LIN {X 0,Y 401.063,Z 357.189,A -85,B 0,C 180,E1 -11072.614,E2 -11072.614} C_VEL
LIN {X 0,Y 401.534,Z 344.039,A -85,B 0,C 180,E1 -11073.183,E2 -11073.183} C_VEL
LIN {X 0,Y 401.795,Z 330.677,A -85,B 0,C 180,E1 -11073.537,E2 -11073.537} C_VEL
LIN {X 0,Y 402.83,Z 248.147,A -85,B 0,C 180,E1 -11075.006,E2 -11075.006} C_VEL
LIN {X 0,Y 398.942,Z 226.266,A -85,B 0,C 180,E1 -11075.573,E2 -11075.573} C_VEL
LIN {X 0,Y 398.046,Z 222.975,A -85,B 0,C 180,E1 -11075.701,E2 -11075.701} C_VEL
LIN {X 0,Y 397.386,Z 219.987,A -85,B 0,C 180,E1 -11076.061,E2 -11076.061} C_VEL
LIN {X 0,Y 397.241,Z 220.003,A -85,B 0,C 180,E1 -11079.163,E2 -11079.163} C_VEL
LIN {X 0,Y 397.225,Z 220.006,A -85,B 0,C 180,E1 -11082.259,E2 -11082.259} C_VEL
LIN {X 0,Y 397.184,Z 220.008,A -85,B 0,C 180,E1 -11085.393,E2 -11085.393} C_VEL
LIN {X 0,Y 397.167,Z 220.014,A -85,B 0,C 180,E1 -11088.574,E2 -11088.574} C_VEL
LIN {X 0,Y 397.102,Z 220.021,A -85,B 0,C 180,E1 -11091.819,E2 -11091.819} C_VEL
LIN {X 0,Y 397.11,Z 220.018,A -85,B 0,C 180,E1 -11095.136,E2 -11095.136} C_VEL
LIN {X 0,Y 397.071,Z 220.024,A -85,B 0,C 180,E1 -11098.549,E2 -11098.549} C_VEL
LIN {X 0,Y 397.086,Z 220.023,A -85,B 0,C 180,E1 -11101.836,E2 -11101.836} C_VEL
LIN {X 0,Y 397.123,Z 220.017,A -85,B 0,C 180,E1 -11104.495,E2 -11104.495} C_VEL
LIN {X 0,Y 397.093,Z 220.021,A -85,B 0,C 180,E1 -11108.277,E2 -11108.277} C_VEL
LIN {X 0,Y 397.056,Z 220.027,A -85,B 0,C 180,E1 -11111.976,E2 -11111.976} C_VEL
LIN {X 0,Y 397.09,Z 220.023,A -85,B 0,C 180,E1 -11115.07,E2 -11115.07} C_VEL
LIN {X 0,Y 397.056,Z 220.025,A -85,B 0,C 180,E1 -11118.024,E2 -11118.024} C_VEL
LIN {X 0,Y 397.092,Z 220.023,A -85,B 0,C 180,E1 -11121.147,E2 -11121.147} C_VEL
LIN {X 0,Y 397.095,Z 220.021,A -85,B 0,C 180,E1 -11124.503,E2 -11124.503} C_VEL
LIN {X 0,Y 397.077,Z 220.022,A -85,B 0,C 180,E1 -11127.928,E2 -11127.928} C_VEL
LIN {X 0,Y 397.119,Z 220.018,A -85,B 0,C 180,E1 -11130.295,E2 -11130.295} C_VEL
LIN {X 0,Y 397.076,Z 220.022,A -85,B 0,C 180,E1 -11133.737,E2 -11133.737} C_VEL
LIN {X 0,Y 397.16,Z 220.084,A -85,B 0,C 180,E1 -11137.363,E2 -11137.363} C_VEL
LIN {X 0,Y 398.579,Z 228.682,A -85,B 0,C 180,E1 -11139.62,E2 -11139.62} C_VEL
LIN {X 0,Y 398.602,Z 228.95,A -85,B 0,C 180,E1 -11139.688,E2 -11139.688} C_VEL
LIN {X 0,Y 402.439,Z 249.604,A -85,B 0,C 180,E1 -11140.323,E2 -11140.323} C_VEL
LIN {X 0,Y 400.599,Z 337.679,A -85,B 0,C 180,E1 -11142.318,E2 -11142.318} C_VEL
LIN {X 0,Y 400.213,Z 351.101,A -85,B 0,C 180,E1 -11142.828,E2 -11142.828} C_VEL
LIN {X 0,Y 399.791,Z 363.98,A -85,B 0,C 180,E1 -11143.533,E2 -11143.533} C_VEL
LIN {X 0,Y 399.118,Z 376.314,A -85,B 0,C 180,E1 -11144.423,E2 -11144.423} C_VEL
LIN {X 0,Y 398.537,Z 387.459,A -85,B 0,C 180,E1 -11145.446,E2 -11145.446} C_VEL
LIN {X 0,Y 397.965,Z 398.566,A -85,B 0,C 180,E1 -11146.727,E2 -11146.727} C_VEL
LIN {X 0,Y 397.414,Z 407.599,A -85,B 0,C 180,E1 -11148.007,E2 -11148.007} C_VEL
LIN {X 0,Y 396.89,Z 416.341,A -85,B 0,C 180,E1 -11149.542,E2 -11149.542} C_VEL
LIN {X 0,Y 396.494,Z 423.36,A -85,B 0,C 180,E1 -11151.077,E2 -11151.077} C_VEL
LIN {X 0,Y 396.215,Z 429.747,A -85,B 0,C 180,E1 -11152.867,E2 -11152.867} C_VEL
LIN {X 0,Y 396.072,Z 433.874,A -85,B 0,C 180,E1 -11154.399,E2 -11154.399} C_VEL
LIN {X 0,Y 395.924,Z 436.902,A -85,B 0,C 180,E1 -11155.928,E2 -11155.928} C_VEL
LIN {X 0,Y 395.946,Z 438.34,A -85,B 0,C 180,E1 -11156.947,E2 -11156.947} C_VEL
LIN {X 0,Y 395.921,Z 439.365,A -85,B 0,C 180,E1 -11157.965,E2 -11157.965} C_VEL
LIN {X 0,Y 395.851,Z 439.942,A -85,B 0,C 180,E1 -11158.982,E2 -11158.982} C_VEL
LIN {X 0,Y 395.86,Z 440.071,A -85,B 0,C 180,E1 -11160,E2 -11160} C_VEL
LIN {X 0,Y 395.915,Z 439.79,A -85,B 0,C 180,E1 -11161.017,E2 -11161.017} C_VEL
LIN {X 0,Y 396.011,Z 439.092,A -85,B 0,C 180,E1 -11162.034,E2 -11162.034} C_VEL
LIN {X 0,Y 396.188,Z 437.92,A -85,B 0,C 180,E1 -11163.05,E2 -11163.05} C_VEL
LIN {X 0,Y 396.462,Z 435.363,A -85,B 0,C 180,E1 -11164.575,E2 -11164.575} C_VEL
LIN {X 0,Y 396.56,Z 431.768,A -85,B 0,C 180,E1 -11166.104,E2 -11166.104} C_VEL
LIN {X 0,Y 397.232,Z 426.428,A -85,B 0,C 180,E1 -11167.782,E2 -11167.782} C_VEL
LIN {X 0,Y 397.81,Z 419.827,A -85,B 0,C 180,E1 -11169.405,E2 -11169.405} C_VEL
LIN {X 0,Y 398.625,Z 411.939,A -85,B 0,C 180,E1 -11170.925,E2 -11170.925} C_VEL
LIN {X 0,Y 399.377,Z 403.929,A -85,B 0,C 180,E1 -11172.191,E2 -11172.191} C_VEL
LIN {X 0,Y 400.233,Z 394.193,A -85,B 0,C 180,E1 -11173.454,E2 -11173.454} C_VEL
LIN {X 0,Y 401.25,Z 383.309,A -85,B 0,C 180,E1 -11174.583,E2 -11174.583} C_VEL
LIN {X 0,Y 402.03,Z 372.326,A -85,B 0,C 180,E1 -11175.504,E2 -11175.504} C_VEL
LIN {X 0,Y 402.835,Z 360.204,A -85,B 0,C 180,E1 -11176.299,E2 -11176.299} C_VEL
LIN {X 0,Y 403.424,Z 346.397,A -85,B 0,C 180,E1 -11176.965,E2 -11176.965} C_VEL
LIN {X 0,Y 403.901,Z 332.803,A -85,B 0,C 180,E1 -11177.401,E2 -11177.401} C_VEL
LIN {X 0,Y 406.565,Z 263.883,A -85,B 0,C 180,E1 -11179.143,E2 -11179.143} C_VEL
LIN {X 0,Y 406.93,Z 252.02,A -85,B 0,C 180,E1 -11179.466,E2 -11179.466} C_VEL
LIN {X 0,Y 404.708,Z 243.879,A -85,B 0,C 180,E1 -11179.902,E2 -11179.902} C_VEL
LIN {X 0,Y 401.099,Z 235.68,A -85,B 0,C 180,E1 -11180.482,E2 -11180.482} C_VEL
LIN {X 0,Y 400.343,Z 233.798,A -85,B 0,C 180,E1 -11180.618,E2 -11180.618} C_VEL
LIN {X 0,Y 398.311,Z 224.634,A -85,B 0,C 180,E1 -11183.943,E2 -11183.943} C_VEL
LIN {X 0,Y 397.149,Z 220.017,A -85,B 0,C 180,E1 -11185.833,E2 -11185.833} C_VEL
LIN {X 0,Y 397.128,Z 220.019,A -85,B 0,C 180,E1 -11188.543,E2 -11188.543} C_VEL
LIN {X 0,Y 397.084,Z 220.024,A -85,B 0,C 180,E1 -11192.071,E2 -11192.071} C_VEL
LIN {X 0,Y 397.125,Z 220.018,A -85,B 0,C 180,E1 -11195.503,E2 -11195.503} C_VEL
LIN {X 0,Y 397.135,Z 220.015,A -85,B 0,C 180,E1 -11198.861,E2 -11198.861} C_VEL
LIN {X 0,Y 397.073,Z 220.024,A -85,B 0,C 180,E1 -11202.267,E2 -11202.267} C_VEL
LIN {X 0,Y 397.091,Z 220.021,A -85,B 0,C 180,E1 -11205.068,E2 -11205.068} C_VEL
LIN {X 0,Y 397.067,Z 220.025,A -85,B 0,C 180,E1 -11208.021,E2 -11208.021} C_VEL
LIN {X 0,Y 397.128,Z 220.016,A -85,B 0,C 180,E1 -11211.139,E2 -11211.139} C_VEL
LIN {X 0,Y 397.123,Z 220.019,A -85,B 0,C 180,E1 -11214.496,E2 -11214.496} C_VEL
LIN {X 0,Y 397.114,Z 220.1,A -85,B 0,C 180,E1 -11217.481,E2 -11217.481} C_VEL
LIN {X 0,Y 399.599,Z 229.04,A -85,B 0,C 180,E1 -11220.497,E2 -11220.497} C_VEL
LIN {X 0,Y 401.612,Z 238.359,A -85,B 0,C 180,E1 -11223.186,E2 -11223.186} C_VEL
LIN {X 0,Y 402.307,Z 242.854,A -85,B 0,C 180,E1 -11224.381,E2 -11224.381} C_VEL
LIN {X 0,Y 400.576,Z 257.062,A -85,B 0,C 180,E1 -11227.566,E2 -11227.566} C_VEL
LIN {X 0,Y 400.165,Z 260.831,A -85,B 0,C 180,E1 -11228.382,E2 -11228.382} C_VEL
LIN {X 0,Y 403.739,Z 277.867,A -85,B 0,C 180,E1 -11229.213,E2 -11229.213} C_VEL
LIN {X 0,Y 405.673,Z 291.849,A -85,B 0,C 180,E1 -11229.776,E2 -11229.776} C_VEL
LIN {X 0,Y 405.744,Z 299.247,A -85,B 0,C 180,E1 -11229.996,E2 -11229.996} C_VEL
LIN {X 0,Y 403.15,Z 373.349,A -85,B 0,C 180,E1 -11231.875,E2 -11231.875} C_VEL
LIN {X 0,Y 402.379,Z 386.533,A -85,B 0,C 180,E1 -11232.398,E2 -11232.398} C_VEL
LIN {X 0,Y 401.432,Z 398.799,A -85,B 0,C 180,E1 -11233.078,E2 -11233.078} C_VEL
LIN {X 0,Y 400.503,Z 410.917,A -85,B 0,C 180,E1 -11233.955,E2 -11233.955} C_VEL
LIN {X 0,Y 399.499,Z 421.992,A -85,B 0,C 180,E1 -11234.96,E2 -11234.96} C_VEL
LIN {X 0,Y 398.415,Z 433.079,A -85,B 0,C 180,E1 -11236.22,E2 -11236.22} C_VEL
LIN {X 0,Y 397.788,Z 442.22,A -85,B 0,C 180,E1 -11237.5,E2 -11237.5} C_VEL
LIN {X 0,Y 397.011,Z 449.795,A -85,B 0,C 180,E1 -11238.77,E2 -11238.77} C_VEL
LIN {X 0,Y 396.51,Z 457.268,A -85,B 0,C 180,E1 -11240.305,E2 -11240.305} C_VEL
LIN {X 0,Y 396.148,Z 463.253,A -85,B 0,C 180,E1 -11241.84,E2 -11241.84} C_VEL
LIN {X 0,Y 395.896,Z 467.98,A -85,B 0,C 180,E1 -11243.373,E2 -11243.373} C_VEL
LIN {X 0,Y 395.83,Z 471.57,A -85,B 0,C 180,E1 -11244.906,E2 -11244.906} C_VEL
LIN {X 0,Y 395.781,Z 473.371,A -85,B 0,C 180,E1 -11245.926,E2 -11245.926} C_VEL
LIN {X 0,Y 395.766,Z 474.741,A -85,B 0,C 180,E1 -11246.945,E2 -11246.945} C_VEL
LIN {X 0,Y 395.856,Z 475.636,A -85,B 0,C 180,E1 -11247.964,E2 -11247.964} C_VEL
LIN {X 0,Y 395.832,Z 476.09,A -85,B 0,C 180,E1 -11248.982,E2 -11248.982} C_VEL
LIN {X 0,Y 395.832,Z 476.126,A -85,B 0,C 180,E1 -11249.999,E2 -11249.999} C_VEL
LIN {X 0,Y 395.832,Z 475.723,A -85,B 0,C 180,E1 -11251.016,E2 -11251.016} C_VEL
LIN {X 0,Y 395.884,Z 474.843,A -85,B 0,C 180,E1 -11252.034,E2 -11252.034} C_VEL
LIN {X 0,Y 395.804,Z 471.823,A -85,B 0,C 180,E1 -11254.072,E2 -11254.072} C_VEL
LIN {X 0,Y 395.825,Z 468.629,A -85,B 0,C 180,E1 -11255.805,E2 -11255.805} C_VEL
LIN {X 0,Y 396.05,Z 463.765,A -85,B 0,C 180,E1 -11257.647,E2 -11257.647} C_VEL
LIN {X 0,Y 396.396,Z 457.411,A -85,B 0,C 180,E1 -11259.438,E2 -11259.438} C_VEL
LIN {X 0,Y 396.877,Z 450.497,A -85,B 0,C 180,E1 -11260.973,E2 -11260.973} C_VEL
LIN {X 0,Y 397.698,Z 441.836,A -85,B 0,C 180,E1 -11262.501,E2 -11262.501} C_VEL
LIN {X 0,Y 398.48,Z 432.076,A -85,B 0,C 180,E1 -11263.892,E2 -11263.892} C_VEL
LIN {X 0,Y 399.464,Z 421.988,A -85,B 0,C 180,E1 -11265.039,E2 -11265.039} C_VEL
LIN {X 0,Y 400.44,Z 410.878,A -85,B 0,C 180,E1 -11266.046,E2 -11266.046} C_VEL
LIN {X 0,Y 401.396,Z 398.415,A -85,B 0,C 180,E1 -11266.922,E2 -11266.922} C_VEL
LIN {X 0,Y 402.198,Z 385.528,A -85,B 0,C 180,E1 -11267.575,E2 -11267.575} C_VEL
LIN {X 0,Y 402.857,Z 372.832,A -85,B 0,C 180,E1 -11268.004,E2 -11268.004} C_VEL
LIN {X 0,Y 403.564,Z 325.155,A -85,B 0,C 180,E1 -11268.907,E2 -11268.907} C_VEL
LIN {X 0,Y 403.921,Z 293.473,A -85,B 0,C 180,E1 -11269.491,E2 -11269.491} C_VEL
LIN {X 0,Y 400.513,Z 269.928,A -85,B 0,C 180,E1 -11270.146,E2 -11270.146} C_VEL
LIN {X 0,Y 398.784,Z 259.631,A -85,B 0,C 180,E1 -11270.458,E2 -11270.458} C_VEL
LIN {X 0,Y 400.229,Z 239.999,A -85,B 0,C 180,E1 -11274.394,E2 -11274.394} C_VEL
LIN {X 0,Y 400.31,Z 236.077,A -85,B 0,C 180,E1 -11275.196,E2 -11275.196} C_VEL
LIN {X 0,Y 397.701,Z 222.504,A -85,B 0,C 180,E1 -11278.168,E2 -11278.168} C_VEL
LIN {X 0,Y 397.184,Z 220.012,A -85,B 0,C 180,E1 -11278.754,E2 -11278.754} C_VEL
LIN {X 0,Y 397.075,Z 220.011,A -85,B 0,C 180,E1 -11282.07,E2 -11282.07} C_VEL
LIN {X 0,Y 397.114,Z 220.009,A -85,B 0,C 180,E1 -11285.502,E2 -11285.502} C_VEL
LIN {X 0,Y 397.087,Z 220.014,A -85,B 0,C 180,E1 -11288.854,E2 -11288.854} C_VEL
LIN {X 0,Y 397.055,Z 220.02,A -85,B 0,C 180,E1 -11292.267,E2 -11292.267} C_VEL
LIN {X 0,Y 397.079,Z 220.02,A -85,B 0,C 180,E1 -11295.068,E2 -11295.068} C_VEL
LIN {X 0,Y 397.046,Z 220.014,A -85,B 0,C 180,E1 -11298.022,E2 -11298.022} C_VEL
LIN {X 0,Y 397.085,Z 220.02,A -85,B 0,C 180,E1 -11301.723,E2 -11301.723} C_VEL
LIN {X 0,Y 397.117,Z 220.01,A -85,B 0,C 180,E1 -11305.506,E2 -11305.506} C_VEL
LIN {X 0,Y 397.069,Z 220.014,A -85,B 0,C 180,E1 -11309.117,E2 -11309.117} C_VEL
LIN {X 0,Y 397.054,Z 220.013,A -85,B 0,C 180,E1 -11312.251,E2 -11312.251} C_VEL
LIN {X 0,Y 397.093,Z 220.02,A -85,B 0,C 180,E1 -11314.864,E2 -11314.864} C_VEL
LIN {X 0,Y 397.085,Z 219.996,A -85,B 0,C 180,E1 -11318.181,E2 -11318.181} C_VEL
LIN {X 0,Y 397.147,Z 220.011,A -85,B 0,C 180,E1 -11321.426,E2 -11321.426} C_VEL
LIN {X 0,Y 397.159,Z 219.999,A -85,B 0,C 180,E1 -11324.607,E2 -11324.607} C_VEL
LIN {X 0,Y 397.209,Z 219.995,A -85,B 0,C 180,E1 -11327.742,E2 -11327.742} C_VEL
LIN {X 0,Y 397.225,Z 220.004,A -85,B 0,C 180,E1 -11330.838,E2 -11330.838} C_VEL
LIN {X 0,Y 397.306,Z 219.977,A -85,B 0,C 180,E1 -11333.908,E2 -11333.908} C_VEL
LIN {X 0,Y 397.437,Z 219.974,A -85,B 0,C 180,E1 -11337.973,E2 -11337.973} C_VEL
LIN {X 0,Y 397.364,Z 219.974,A -85,B 0,C 180,E1 -11341.014,E2 -11341.014} C_VEL
LIN {X 0,Y 397.321,Z 219.969,A -85,B 0,C 180,E1 -11343.042,E2 -11343.042} C_VEL
LIN {X 0,Y 397.334,Z 219.985,A -85,B 0,C 180,E1 -11346.643,E2 -11346.643} C_VEL
LIN {X 0,Y 397.244,Z 219.989,A -85,B 0,C 180,E1 -11349.162,E2 -11349.162} C_VEL
LIN {X 0,Y 397.21,Z 220,A -85,B 0,C 180,E1 -11352.259,E2 -11352.259} C_VEL
LIN {X 0,Y 397.171,Z 220.008,A -85,B 0,C 180,E1 -11355.393,E2 -11355.393} C_VEL
LIN {X 0,Y 397.15,Z 220.005,A -85,B 0,C 180,E1 -11358.574,E2 -11358.574} C_VEL
LIN {X 0,Y 397.102,Z 220.017,A -85,B 0,C 180,E1 -11361.819,E2 -11361.819} C_VEL
LIN {X 0,Y 397.146,Z 220.011,A -85,B 0,C 180,E1 -11365.513,E2 -11365.513} C_VEL
LIN {X 0,Y 397.116,Z 220.011,A -85,B 0,C 180,E1 -11368.545,E2 -11368.545} C_VEL
LIN {X 0,Y 397.073,Z 220.023,A -85,B 0,C 180,E1 -11372.073,E2 -11372.073} C_VEL
LIN {X 0,Y 397.115,Z 220.021,A -85,B 0,C 180,E1 -11375.505,E2 -11375.505} C_VEL
LIN {X 0,Y 397.129,Z 220.013,A -85,B 0,C 180,E1 -11378.863,E2 -11378.863} C_VEL
LIN {X 0,Y 397.067,Z 220.019,A -85,B 0,C 180,E1 -11382.268,E2 -11382.268} C_VEL
LIN {X 0,Y 397.088,Z 220.02,A -85,B 0,C 180,E1 -11385.069,E2 -11385.069} C_VEL
LIN {X 0,Y 397.065,Z 220.022,A -85,B 0,C 180,E1 -11388.022,E2 -11388.022} C_VEL
LIN {X 0,Y 397.129,Z 220.017,A -85,B 0,C 180,E1 -11391.14,E2 -11391.14} C_VEL
LIN {X 0,Y 397.189,Z 220.178,A -85,B 0,C 180,E1 -11394.835,E2 -11394.835} C_VEL
LIN {X 0,Y 398.26,Z 223.723,A -85,B 0,C 180,E1 -11395.233,E2 -11395.233} C_VEL
LIN {X 0,Y 402.441,Z 234.001,A -85,B 0,C 180,E1 -11395.7,E2 -11395.7} C_VEL
LIN {X 0,Y 405.169,Z 249.064,A -85,B 0,C 180,E1 -11396.158,E2 -11396.158} C_VEL
LIN {X 0,Y 403.759,Z 336.274,A -85,B 0,C 180,E1 -11397.751,E2 -11397.751} C_VEL
LIN {X 0,Y 403.309,Z 349.643,A -85,B 0,C 180,E1 -11398.19,E2 -11398.19} C_VEL
LIN {X 0,Y 402.684,Z 362.586,A -85,B 0,C 180,E1 -11398.845,E2 -11398.845} C_VEL
LIN {X 0,Y 401.924,Z 374.716,A -85,B 0,C 180,E1 -11399.676,E2 -11399.676} C_VEL
LIN {X 0,Y 400.96,Z 386.467,A -85,B 0,C 180,E1 -11400.728,E2 -11400.728} C_VEL
LIN {X 0,Y 399.92,Z 397.351,A -85,B 0,C 180,E1 -11401.961,E2 -11401.961} C_VEL
LIN {X 0,Y 399.022,Z 406.833,A -85,B 0,C 180,E1 -11403.313,E2 -11403.313} C_VEL
LIN {X 0,Y 398.081,Z 415.911,A -85,B 0,C 180,E1 -11404.932,E2 -11404.932} C_VEL
LIN {X 0,Y 397.365,Z 423.026,A -85,B 0,C 180,E1 -11406.539,E2 -11406.539} C_VEL
LIN {X 0,Y 396.787,Z 428.692,A -85,B 0,C 180,E1 -11408.165,E2 -11408.165} C_VEL
LIN {X 0,Y 396.333,Z 433.595,A -85,B 0,C 180,E1 -11410.024,E2 -11410.024} C_VEL
LIN {X 0,Y 396.04,Z 436.166,A -85,B 0,C 180,E1 -11411.373,E2 -11411.373} C_VEL
LIN {X 0,Y 395.884,Z 437.703,A -85,B 0,C 180,E1 -11412.436,E2 -11412.436} C_VEL
LIN {X 0,Y 395.822,Z 438.749,A -85,B 0,C 180,E1 -11413.497,E2 -11413.497} C_VEL
LIN {X 0,Y 395.754,Z 439.384,A -85,B 0,C 180,E1 -11414.552,E2 -11414.552} C_VEL
LIN {X 0,Y 395.717,Z 439.618,A -85,B 0,C 180,E1 -11415.604,E2 -11415.604} C_VEL
LIN {X 0,Y 395.783,Z 438.843,A -85,B 0,C 180,E1 -11417.595,E2 -11417.595} C_VEL
LIN {X 0,Y 395.809,Z 437.743,A -85,B 0,C 180,E1 -11418.738,E2 -11418.738} C_VEL
LIN {X 0,Y 395.835,Z 436.284,A -85,B 0,C 180,E1 -11419.774,E2 -11419.774} C_VEL
LIN {X 0,Y 396.083,Z 433.264,A -85,B 0,C 180,E1 -11421.327,E2 -11421.327} C_VEL
LIN {X 0,Y 396.402,Z 428.325,A -85,B 0,C 180,E1 -11423.15,E2 -11423.15} C_VEL
LIN {X 0,Y 396.707,Z 421.962,A -85,B 0,C 180,E1 -11424.919,E2 -11424.919} C_VEL
LIN {X 0,Y 397.295,Z 414.866,A -85,B 0,C 180,E1 -11426.451,E2 -11426.451} C_VEL
LIN {X 0,Y 397.977,Z 406.078,A -85,B 0,C 180,E1 -11427.977,E2 -11427.977} C_VEL
LIN {X 0,Y 398.722,Z 395.987,A -85,B 0,C 180,E1 -11429.37,E2 -11429.37} C_VEL
LIN {X 0,Y 399.486,Z 385.754,A -85,B 0,C 180,E1 -11430.505,E2 -11430.505} C_VEL
LIN {X 0,Y 400.238,Z 374.372,A -85,B 0,C 180,E1 -11431.51,E2 -11431.51} C_VEL
LIN {X 0,Y 400.524,Z 369.63,A -85,B 0,C 180,E1 -11431.859,E2 -11431.859} C_VEL
LIN {X 0,Y 400.19,Z 364.343,A -85,B 0,C 180,E1 -11432.233,E2 -11432.233} C_VEL
LIN {X 0,Y 397.799,Z 355.633,A -85,B 0,C 180,E1 -11432.82,E2 -11432.82} C_VEL
LIN {X 0,Y 395.32,Z 346.674,A -85,B 0,C 180,E1 -11433.318,E2 -11433.318} C_VEL
LIN {X 0,Y 394.766,Z 340.998,A -85,B 0,C 180,E1 -11433.539,E2 -11433.539} C_VEL
LIN {X 0,Y 395.025,Z 326.392,A -85,B 0,C 180,E1 -11433.876,E2 -11433.876} C_VEL
LIN {X 0,Y 395.954,Z 248.651,A -85,B 0,C 180,E1 -11435.284,E2 -11435.284} C_VEL
LIN {X 0,Y 392.347,Z 228.274,A -85,B 0,C 180,E1 -11435.822,E2 -11435.822} C_VEL
LIN {X 0,Y 390.875,Z 223.251,A -85,B 0,C 180,E1 -11436,E2 -11436} C_VEL
LIN {X 0,Y 390.309,Z 220.868,A -85,B 0,C 180,E1 -11436.268,E2 -11436.268} C_VEL
LIN {X 0,Y 390.198,Z 220.879,A -85,B 0,C 180,E1 -11439.33,E2 -11439.33} C_VEL
LIN {X 0,Y 390.176,Z 220.884,A -85,B 0,C 180,E1 -11442.484,E2 -11442.484} C_VEL
LIN {X 0,Y 390.145,Z 220.885,A -85,B 0,C 180,E1 -11445.678,E2 -11445.678} C_VEL
LIN {X 0,Y 390.111,Z 220.89,A -85,B 0,C 180,E1 -11448.923,E2 -11448.923} C_VEL
LIN {X 0,Y 390.042,Z 220.901,A -85,B 0,C 180,E1 -11452.235,E2 -11452.235} C_VEL
LIN {X 0,Y 390.056,Z 220.899,A -85,B 0,C 180,E1 -11455.723,E2 -11455.723} C_VEL
LIN {X 0,Y 390.031,Z 220.899,A -85,B 0,C 180,E1 -11459.113,E2 -11459.113} C_VEL
LIN {X 0,Y 390.047,Z 220.897,A -85,B 0,C 180,E1 -11462.722,E2 -11462.722} C_VEL
LIN {X 0,Y 390.049,Z 220.9,A -85,B 0,C 180,E1 -11465.823,E2 -11465.823} C_VEL
LIN {X 0,Y 390.04,Z 220.9,A -85,B 0,C 180,E1 -11469.212,E2 -11469.212} C_VEL
LIN {X 0,Y 390.035,Z 220.899,A -85,B 0,C 180,E1 -11472.372,E2 -11472.372} C_VEL
LIN {X 0,Y 390.046,Z 220.901,A -85,B 0,C 180,E1 -11475.354,E2 -11475.354} C_VEL
LIN {X 0,Y 390.019,Z 220.901,A -85,B 0,C 180,E1 -11478.185,E2 -11478.185} C_VEL
LIN {X 0,Y 390.059,Z 220.899,A -85,B 0,C 180,E1 -11480.903,E2 -11480.903} C_VEL
LIN {X 0,Y 390.066,Z 220.898,A -85,B 0,C 180,E1 -11484.791,E2 -11484.791} C_VEL
LIN {X 0,Y 390.031,Z 220.899,A -85,B 0,C 180,E1 -11487.878,E2 -11487.878} C_VEL
LIN {X 0,Y 390.027,Z 220.903,A -85,B 0,C 180,E1 -11490.887,E2 -11490.887} C_VEL
LIN {X 0,Y 390.067,Z 220.897,A -85,B 0,C 180,E1 -11494.378,E2 -11494.378} C_VEL
LIN {X 0,Y 390.108,Z 220.937,A -85,B 0,C 180,E1 -11497.211,E2 -11497.211} C_VEL
LIN {X 0,Y 391.556,Z 229.176,A -85,B 0,C 180,E1 -11499.409,E2 -11499.409} C_VEL
LIN {X 0,Y 395.558,Z 250.268,A -85,B 0,C 180,E1 -11500.09,E2 -11500.09} C_VEL
LIN {X 0,Y 393.638,Z 337.821,A -85,B 0,C 180,E1 -11502.129,E2 -11502.129} C_VEL
LIN {X 0,Y 393.23,Z 351.232,A -85,B 0,C 180,E1 -11502.647,E2 -11502.647} C_VEL
LIN {X 0,Y 392.788,Z 364.143,A -85,B 0,C 180,E1 -11503.364,E2 -11503.364} C_VEL
LIN {X 0,Y 392.107,Z 376.495,A -85,B 0,C 180,E1 -11504.27,E2 -11504.27} C_VEL
LIN {X 0,Y 391.519,Z 387.674,A -85,B 0,C 180,E1 -11505.312,E2 -11505.312} C_VEL
LIN {X 0,Y 390.93,Z 398.804,A -85,B 0,C 180,E1 -11506.617,E2 -11506.617} C_VEL
LIN {X 0,Y 390.296,Z 408.668,A -85,B 0,C 180,E1 -11508.048,E2 -11508.048} C_VEL
LIN {X 0,Y 389.793,Z 417.273,A -85,B 0,C 180,E1 -11509.612,E2 -11509.612} C_VEL
LIN {X 0,Y 389.392,Z 424.199,A -85,B 0,C 180,E1 -11511.175,E2 -11511.175} C_VEL
LIN {X 0,Y 389.131,Z 429.692,A -85,B 0,C 180,E1 -11512.737,E2 -11512.737} C_VEL
LIN {X 0,Y 388.998,Z 433.93,A -85,B 0,C 180,E1 -11514.297,E2 -11514.297} C_VEL
LIN {X 0,Y 388.846,Z 437.056,A -85,B 0,C 180,E1 -11515.854,E2 -11515.854} C_VEL
LIN {X 0,Y 388.847,Z 438.54,A -85,B 0,C 180,E1 -11516.892,E2 -11516.892} C_VEL
LIN {X 0,Y 388.837,Z 439.608,A -85,B 0,C 180,E1 -11517.928,E2 -11517.928} C_VEL
LIN {X 0,Y 388.78,Z 440.262,A -85,B 0,C 180,E1 -11518.964,E2 -11518.964} C_VEL
LIN {X 0,Y 388.785,Z 440.443,A -85,B 0,C 180,E1 -11520,E2 -11520} C_VEL
LIN {X 0,Y 388.841,Z 440.204,A -85,B 0,C 180,E1 -11521.035,E2 -11521.035} C_VEL
LIN {X 0,Y 388.945,Z 439.556,A -85,B 0,C 180,E1 -11522.071,E2 -11522.071} C_VEL
LIN {X 0,Y 389.131,Z 438.453,A -85,B 0,C 180,E1 -11523.106,E2 -11523.106} C_VEL
LIN {X 0,Y 389.328,Z 436.899,A -85,B 0,C 180,E1 -11524.141,E2 -11524.141} C_VEL
LIN {X 0,Y 389.551,Z 433.741,A -85,B 0,C 180,E1 -11525.694,E2 -11525.694} C_VEL
LIN {X 0,Y 389.97,Z 429.466,A -85,B 0,C 180,E1 -11527.247,E2 -11527.247} C_VEL
LIN {X 0,Y 390.591,Z 423.97,A -85,B 0,C 180,E1 -11528.797,E2 -11528.797} C_VEL
LIN {X 0,Y 391.311,Z 417.093,A -85,B 0,C 180,E1 -11530.346,E2 -11530.346} C_VEL
LIN {X 0,Y 392.176,Z 408.454,A -85,B 0,C 180,E1 -11531.893,E2 -11531.893} C_VEL
LIN {X 0,Y 393.015,Z 399.655,A -85,B 0,C 180,E1 -11533.179,E2 -11533.179} C_VEL
LIN {X 0,Y 394.111,Z 388.807,A -85,B 0,C 180,E1 -11534.457,E2 -11534.457} C_VEL
LIN {X 0,Y 395.183,Z 376.959,A -85,B 0,C 180,E1 -11535.561,E2 -11535.561} C_VEL
LIN {X 0,Y 395.965,Z 365.858,A -85,B 0,C 180,E1 -11536.387,E2 -11536.387} C_VEL
LIN {X 0,Y 396.725,Z 353.478,A -85,B 0,C 180,E1 -11537.088,E2 -11537.088} C_VEL
LIN {X 0,Y 397.307,Z 341.008,A -85,B 0,C 180,E1 -11537.6,E2 -11537.6} C_VEL
LIN {X 0,Y 398.13,Z 317.692,A -85,B 0,C 180,E1 -11538.227,E2 -11538.227} C_VEL
LIN {X 0,Y 400.857,Z 253.841,A -85,B 0,C 180,E1 -11539.925,E2 -11539.925} C_VEL
LIN {X 0,Y 398.802,Z 246.292,A -85,B 0,C 180,E1 -11540.35,E2 -11540.35} C_VEL
LIN {X 0,Y 394.609,Z 237.226,A -85,B 0,C 180,E1 -11541.048,E2 -11541.048} C_VEL
LIN {X 0,Y 393.316,Z 234.43,A -85,B 0,C 180,E1 -11541.279,E2 -11541.279} C_VEL
LIN {X 0,Y 391.488,Z 226.244,A -85,B 0,C 180,E1 -11544.387,E2 -11544.387} C_VEL
LIN {X 0,Y 390.119,Z 220.893,A -85,B 0,C 180,E1 -11546.768,E2 -11546.768} C_VEL
LIN {X 0,Y 390.045,Z 220.902,A -85,B 0,C 180,E1 -11550.299,E2 -11550.299} C_VEL
LIN {X 0,Y 390.074,Z 220.897,A -85,B 0,C 180,E1 -11554.024,E2 -11554.024} C_VEL
LIN {X 0,Y 390.048,Z 220.899,A -85,B 0,C 180,E1 -11557.55,E2 -11557.55} C_VEL
LIN {X 0,Y 390.061,Z 220.896,A -85,B 0,C 180,E1 -11560.821,E2 -11560.821} C_VEL
LIN {X 0,Y 390.059,Z 220.898,A -85,B 0,C 180,E1 -11563.885,E2 -11563.885} C_VEL
LIN {X 0,Y 390.06,Z 220.896,A -85,B 0,C 180,E1 -11566.789,E2 -11566.789} C_VEL
LIN {X 0,Y 390.06,Z 220.898,A -85,B 0,C 180,E1 -11569.56,E2 -11569.56} C_VEL
LIN {X 0,Y 390.046,Z 220.9,A -85,B 0,C 180,E1 -11572.449,E2 -11572.449} C_VEL
LIN {X 0,Y 390.073,Z 220.899,A -85,B 0,C 180,E1 -11575.975,E2 -11575.975} C_VEL
LIN {X 0,Y 390.084,Z 220.984,A -85,B 0,C 180,E1 -11576.588,E2 -11576.588} C_VEL
LIN {X 0,Y 392.667,Z 230.248,A -85,B 0,C 180,E1 -11579.923,E2 -11579.923} C_VEL
LIN {X 0,Y 394.511,Z 238.32,A -85,B 0,C 180,E1 -11582.407,E2 -11582.407} C_VEL
LIN {X 0,Y 395.605,Z 244.786,A -85,B 0,C 180,E1 -11584.198,E2 -11584.198} C_VEL
LIN {X 0,Y 393.724,Z 259.088,A -85,B 0,C 180,E1 -11587.486,E2 -11587.486} C_VEL
LIN {X 0,Y 393.579,Z 260.496,A -85,B 0,C 180,E1 -11587.774,E2 -11587.774} C_VEL
LIN {X 0,Y 397.367,Z 277.912,A -85,B 0,C 180,E1 -11588.68,E2 -11588.68} C_VEL
LIN {X 0,Y 399.363,Z 292.156,A -85,B 0,C 180,E1 -11589.287,E2 -11589.287} C_VEL
LIN {X 0,Y 399.531,Z 298.099,A -85,B 0,C 180,E1 -11589.482,E2 -11589.482} C_VEL
LIN {X 0,Y 396.683,Z 372.644,A -85,B 0,C 180,E1 -11591.436,E2 -11591.436} C_VEL
LIN {X 0,Y 395.862,Z 385.791,A -85,B 0,C 180,E1 -11591.965,E2 -11591.965} C_VEL
LIN {X 0,Y 394.891,Z 398.076,A -85,B 0,C 180,E1 -11592.655,E2 -11592.655} C_VEL
LIN {X 0,Y 393.841,Z 410.216,A -85,B 0,C 180,E1 -11593.542,E2 -11593.542} C_VEL
LIN {X 0,Y 392.808,Z 421.315,A -85,B 0,C 180,E1 -11594.564,E2 -11594.564} C_VEL
LIN {X 0,Y 391.587,Z 432.92,A -85,B 0,C 180,E1 -11595.905,E2 -11595.905} C_VEL
LIN {X 0,Y 390.852,Z 442.456,A -85,B 0,C 180,E1 -11597.274,E2 -11597.274} C_VEL
LIN {X 0,Y 389.911,Z 451.231,A -85,B 0,C 180,E1 -11598.826,E2 -11598.826} C_VEL
LIN {X 0,Y 389.397,Z 458.346,A -85,B 0,C 180,E1 -11600.388,E2 -11600.388} C_VEL
LIN {X 0,Y 389.004,Z 464.891,A -85,B 0,C 180,E1 -11602.211,E2 -11602.211} C_VEL
LIN {X 0,Y 388.751,Z 469.421,A -85,B 0,C 180,E1 -11603.887,E2 -11603.887} C_VEL
LIN {X 0,Y 388.704,Z 473.153,A -85,B 0,C 180,E1 -11605.851,E2 -11605.851} C_VEL
LIN {X 0,Y 388.669,Z 474.478,A -85,B 0,C 180,E1 -11606.889,E2 -11606.889} C_VEL
LIN {X 0,Y 388.754,Z 475.329,A -85,B 0,C 180,E1 -11607.927,E2 -11607.927} C_VEL
LIN {X 0,Y 388.761,Z 475.757,A -85,B 0,C 180,E1 -11608.963,E2 -11608.963} C_VEL
LIN {X 0,Y 388.758,Z 475.762,A -85,B 0,C 180,E1 -11609.999,E2 -11609.999} C_VEL
LIN {X 0,Y 388.762,Z 475.296,A -85,B 0,C 180,E1 -11611.035,E2 -11611.035} C_VEL
LIN {X 0,Y 388.816,Z 474.382,A -85,B 0,C 180,E1 -11612.071,E2 -11612.071} C_VEL
LIN {X 0,Y 388.727,Z 471.581,A -85,B 0,C 180,E1 -11614.146,E2 -11614.146} C_VEL
LIN {X 0,Y 388.762,Z 469.879,A -85,B 0,C 180,E1 -11615.185,E2 -11615.185} C_VEL
LIN {X 0,Y 388.816,Z 466.475,A -85,B 0,C 180,E1 -11616.746,E2 -11616.746} C_VEL
LIN {X 0,Y 389.077,Z 461.986,A -85,B 0,C 180,E1 -11618.307,E2 -11618.307} C_VEL
LIN {X 0,Y 389.527,Z 455.167,A -85,B 0,C 180,E1 -11620.131,E2 -11620.131} C_VEL
LIN {X 0,Y 390.171,Z 447.771,A -85,B 0,C 180,E1 -11621.69,E2 -11621.69} C_VEL
LIN {X 0,Y 390.946,Z 440.241,A -85,B 0,C 180,E1 -11622.985,E2 -11622.985} C_VEL
LIN {X 0,Y 391.773,Z 430.389,A -85,B 0,C 180,E1 -11624.372,E2 -11624.372} C_VEL
LIN {X 0,Y 392.861,Z 419.683,A -85,B 0,C 180,E1 -11625.564,E2 -11625.564} C_VEL
LIN {X 0,Y 393.923,Z 408.134,A -85,B 0,C 180,E1 -11626.585,E2 -11626.585} C_VEL
LIN {X 0,Y 394.882,Z 395.807,A -85,B 0,C 180,E1 -11627.41,E2 -11627.41} C_VEL
LIN {X 0,Y 395.696,Z 383.581,A -85,B 0,C 180,E1 -11628.007,E2 -11628.007} C_VEL
LIN {X 0,Y 396.301,Z 371.196,A -85,B 0,C 180,E1 -11628.413,E2 -11628.413} C_VEL
LIN {X 0,Y 397.419,Z 294.775,A -85,B 0,C 180,E1 -11629.854,E2 -11629.854} C_VEL
LIN {X 0,Y 394.018,Z 271.108,A -85,B 0,C 180,E1 -11630.528,E2 -11630.528} C_VEL
LIN {X 0,Y 391.855,Z 258.457,A -85,B 0,C 180,E1 -11630.927,E2 -11630.927} C_VEL
LIN {X 0,Y 393.384,Z 239.402,A -85,B 0,C 180,E1 -11634.823,E2 -11634.823} C_VEL
LIN {X 0,Y 392.76,Z 233.995,A -85,B 0,C 180,E1 -11635.987,E2 -11635.987} C_VEL
LIN {X 0,Y 390.142,Z 220.889,A -85,B 0,C 180,E1 -11638.946,E2 -11638.946} C_VEL
LIN {X 0,Y 390.039,Z 220.879,A -85,B 0,C 180,E1 -11642.72,E2 -11642.72} C_VEL
LIN {X 0,Y 390.051,Z 220.892,A -85,B 0,C 180,E1 -11645.824,E2 -11645.824} C_VEL
LIN {X 0,Y 390.031,Z 220.892,A -85,B 0,C 180,E1 -11649.211,E2 -11649.211} C_VEL
LIN {X 0,Y 390.03,Z 220.895,A -85,B 0,C 180,E1 -11652.372,E2 -11652.372} C_VEL
LIN {X 0,Y 390.036,Z 220.9,A -85,B 0,C 180,E1 -11655.353,E2 -11655.353} C_VEL
LIN {X 0,Y 390.009,Z 220.889,A -85,B 0,C 180,E1 -11658.184,E2 -11658.184} C_VEL
LIN {X 0,Y 390.051,Z 220.897,A -85,B 0,C 180,E1 -11660.903,E2 -11660.903} C_VEL
LIN {X 0,Y 390.077,Z 220.878,A -85,B 0,C 180,E1 -11664.792,E2 -11664.792} C_VEL
LIN {X 0,Y 390.015,Z 220.897,A -85,B 0,C 180,E1 -11668.495,E2 -11668.495} C_VEL
LIN {X 0,Y 390.006,Z 220.89,A -85,B 0,C 180,E1 -11672.002,E2 -11672.002} C_VEL
LIN {X 0,Y 390.032,Z 220.891,A -85,B 0,C 180,E1 -11675.516,E2 -11675.516} C_VEL
LIN {X 0,Y 390.046,Z 220.878,A -85,B 0,C 180,E1 -11678.877,E2 -11678.877} C_VEL
LIN {X 0,Y 390.102,Z 220.889,A -85,B 0,C 180,E1 -11682.166,E2 -11682.166} C_VEL
LIN {X 0,Y 390.125,Z 220.866,A -85,B 0,C 180,E1 -11685.392,E2 -11685.392} C_VEL
LIN {X 0,Y 390.135,Z 220.882,A -85,B 0,C 180,E1 -11688.571,E2 -11688.571} C_VEL
LIN {X 0,Y 390.246,Z 220.872,A -85,B 0,C 180,E1 -11692.087,E2 -11692.087} C_VEL
LIN {X 0,Y 390.191,Z 220.859,A -85,B 0,C 180,E1 -11694.833,E2 -11694.833} C_VEL
LIN {X 0,Y 390.404,Z 220.85,A -85,B 0,C 180,E1 -11697.937,E2 -11697.937} C_VEL
LIN {X 0,Y 390.33,Z 220.85,A -85,B 0,C 180,E1 -11701.032,E2 -11701.032} C_VEL
LIN {X 0,Y 390.258,Z 220.849,A -85,B 0,C 180,E1 -11703.097,E2 -11703.097} C_VEL
LIN {X 0,Y 390.29,Z 220.863,A -85,B 0,C 180,E1 -11706.638,E2 -11706.638} C_VEL
LIN {X 0,Y 390.196,Z 220.867,A -85,B 0,C 180,E1 -11709.329,E2 -11709.329} C_VEL
LIN {X 0,Y 390.187,Z 220.877,A -85,B 0,C 180,E1 -11713.439,E2 -11713.439} C_VEL
LIN {X 0,Y 390.121,Z 220.873,A -85,B 0,C 180,E1 -11717.299,E2 -11717.299} C_VEL
LIN {X 0,Y 390.081,Z 220.892,A -85,B 0,C 180,E1 -11720.471,E2 -11720.471} C_VEL
LIN {X 0,Y 390.083,Z 220.883,A -85,B 0,C 180,E1 -11723.352,E2 -11723.352} C_VEL
LIN {X 0,Y 390.107,Z 220.89,A -85,B 0,C 180,E1 -11726.769,E2 -11726.769} C_VEL
LIN {X 0,Y 390.033,Z 220.896,A -85,B 0,C 180,E1 -11730.301,E2 -11730.301} C_VEL
LIN {X 0,Y 390.063,Z 220.888,A -85,B 0,C 180,E1 -11734.026,E2 -11734.026} C_VEL
LIN {X 0,Y 390.041,Z 220.896,A -85,B 0,C 180,E1 -11737.553,E2 -11737.553} C_VEL
LIN {X 0,Y 390.053,Z 220.902,A -85,B 0,C 180,E1 -11740.823,E2 -11740.823} C_VEL
LIN {X 0,Y 390.053,Z 220.898,A -85,B 0,C 180,E1 -11743.888,E2 -11743.888} C_VEL
LIN {X 0,Y 390.056,Z 220.899,A -85,B 0,C 180,E1 -11746.791,E2 -11746.791} C_VEL
LIN {X 0,Y 390.054,Z 220.895,A -85,B 0,C 180,E1 -11749.562,E2 -11749.562} C_VEL
LIN {X 0,Y 390.041,Z 220.901,A -85,B 0,C 180,E1 -11752.451,E2 -11752.451} C_VEL
LIN {X 0,Y 390.084,Z 220.915,A -85,B 0,C 180,E1 -11754.418,E2 -11754.418} C_VEL
LIN {X 0,Y 391.009,Z 223.941,A -85,B 0,C 180,E1 -11754.755,E2 -11754.755} C_VEL
LIN {X 0,Y 396.258,Z 236.649,A -85,B 0,C 180,E1 -11755.356,E2 -11755.356} C_VEL
LIN {X 0,Y 398.682,Z 251.281,A -85,B 0,C 180,E1 -11755.797,E2 -11755.797} C_VEL
LIN {X 0,Y 397.186,Z 336.5,A -85,B 0,C 180,E1 -11757.377,E2 -11757.377} C_VEL
LIN {X 0,Y 396.716,Z 349.901,A -85,B 0,C 180,E1 -11757.822,E2 -11757.822} C_VEL
LIN {X 0,Y 396.1,Z 362.119,A -85,B 0,C 180,E1 -11758.442,E2 -11758.442} C_VEL
LIN {X 0,Y 395.298,Z 374.082,A -85,B 0,C 180,E1 -11759.261,E2 -11759.261} C_VEL
LIN {X 0,Y 394.407,Z 384.977,A -85,B 0,C 180,E1 -11760.219,E2 -11760.219} C_VEL
LIN {X 0,Y 393.406,Z 394.891,A -85,B 0,C 180,E1 -11761.309,E2 -11761.309} C_VEL
LIN {X 0,Y 392.487,Z 404.002,A -85,B 0,C 180,E1 -11762.544,E2 -11762.544} C_VEL
LIN {X 0,Y 391.684,Z 411.571,A -85,B 0,C 180,E1 -11763.787,E2 -11763.787} C_VEL
LIN {X 0,Y 390.857,Z 419.077,A -85,B 0,C 180,E1 -11765.289,E2 -11765.289} C_VEL
LIN {X 0,Y 390.229,Z 424.837,A -85,B 0,C 180,E1 -11766.71,E2 -11766.71} C_VEL
LIN {X 0,Y 389.68,Z 430.017,A -85,B 0,C 180,E1 -11768.303,E2 -11768.303} C_VEL
LIN {X 0,Y 389.271,Z 434.088,A -85,B 0,C 180,E1 -11769.94,E2 -11769.94} C_VEL
LIN {X 0,Y 389.034,Z 436.137,A -85,B 0,C 180,E1 -11771.025,E2 -11771.025} C_VEL
LIN {X 0,Y 388.843,Z 437.746,A -85,B 0,C 180,E1 -11772.107,E2 -11772.107} C_VEL
LIN {X 0,Y 388.761,Z 439.041,A -85,B 0,C 180,E1 -11773.363,E2 -11773.363} C_VEL
LIN {X 0,Y 388.623,Z 439.907,A -85,B 0,C 180,E1 -11775.335,E2 -11775.335} C_VEL
LIN {X 0,Y 388.617,Z 439.8,A -85,B 0,C 180,E1 -11776.404,E2 -11776.404} C_VEL
LIN {X 0,Y 388.704,Z 439.197,A -85,B 0,C 180,E1 -11777.518,E2 -11777.518} C_VEL
LIN {X 0,Y 388.74,Z 436.918,A -85,B 0,C 180,E1 -11779.585,E2 -11779.585} C_VEL
LIN {X 0,Y 388.967,Z 434.028,A -85,B 0,C 180,E1 -11781.167,E2 -11781.167} C_VEL
LIN {X 0,Y 389.228,Z 430.101,A -85,B 0,C 180,E1 -11782.74,E2 -11782.74} C_VEL
LIN {X 0,Y 389.511,Z 425.029,A -85,B 0,C 180,E1 -11784.306,E2 -11784.306} C_VEL
LIN {X 0,Y 390.042,Z 418.618,A -85,B 0,C 180,E1 -11785.868,E2 -11785.868} C_VEL
LIN {X 0,Y 390.58,Z 410.682,A -85,B 0,C 180,E1 -11787.423,E2 -11787.423} C_VEL
LIN {X 0,Y 391.239,Z 402.563,A -85,B 0,C 180,E1 -11788.714,E2 -11788.714} C_VEL
LIN {X 0,Y 392.047,Z 392.6,A -85,B 0,C 180,E1 -11790.001,E2 -11790.001} C_VEL
LIN {X 0,Y 392.906,Z 381.422,A -85,B 0,C 180,E1 -11791.154,E2 -11791.154} C_VEL
LIN {X 0,Y 393.625,Z 369.957,A -85,B 0,C 180,E1 -11792.085,E2 -11792.085} C_VEL
LIN {X 0,Y 394.123,Z 358.297,A -85,B 0,C 180,E1 -11792.812,E2 -11792.812} C_VEL
LIN {X 0,Y 394.642,Z 344.842,A -85,B 0,C 180,E1 -11793.414,E2 -11793.414} C_VEL
LIN {X 0,Y 394.766,Z 340.998,A -85,B 0,C 180,E1 -11793.539,E2 -11793.539} C_VEL
LIN {X 0,Y 394.206,Z 335.251,A -85,B 0,C 180,E1 -11793.729,E2 -11793.729} C_VEL
LIN {X 0,Y 388.878,Z 316.539,A -85,B 0,C 180,E1 -11794.308,E2 -11794.308} C_VEL
LIN {X 0,Y 388.39,Z 310.716,A -85,B 0,C 180,E1 -11794.432,E2 -11794.432} C_VEL
LIN {X 0,Y 389.204,Z 249.875,A -85,B 0,C 180,E1 -11795.55,E2 -11795.55} C_VEL
LIN {X 0,Y 385.643,Z 229.894,A -85,B 0,C 180,E1 -11796.089,E2 -11796.089} C_VEL
LIN {X 0,Y 383.677,Z 223.516,A -85,B 0,C 180,E1 -11796.311,E2 -11796.311} C_VEL
LIN {X 0,Y 383.27,Z 221.744,A -85,B 0,C 180,E1 -11796.516,E2 -11796.516} C_VEL
LIN {X 0,Y 383.149,Z 221.756,A -85,B 0,C 180,E1 -11799.503,E2 -11799.503} C_VEL
LIN {X 0,Y 383.132,Z 221.758,A -85,B 0,C 180,E1 -11803.537,E2 -11803.537} C_VEL
LIN {X 0,Y 383.101,Z 221.762,A -85,B 0,C 180,E1 -11807.455,E2 -11807.455} C_VEL
LIN {X 0,Y 383.035,Z 221.773,A -85,B 0,C 180,E1 -11810.648,E2 -11810.648} C_VEL
LIN {X 0,Y 383.016,Z 221.776,A -85,B 0,C 180,E1 -11813.81,E2 -11813.81} C_VEL
LIN {X 0,Y 382.977,Z 221.778,A -85,B 0,C 180,E1 -11817.309,E2 -11817.309} C_VEL
LIN {X 0,Y 382.987,Z 221.776,A -85,B 0,C 180,E1 -11820.919,E2 -11820.919} C_VEL
LIN {X 0,Y 383.018,Z 221.773,A -85,B 0,C 180,E1 -11824.669,E2 -11824.669} C_VEL
LIN {X 0,Y 382.997,Z 221.779,A -85,B 0,C 180,E1 -11827.902,E2 -11827.902} C_VEL
LIN {X 0,Y 382.966,Z 221.783,A -85,B 0,C 180,E1 -11831.351,E2 -11831.351} C_VEL
LIN {X 0,Y 382.994,Z 221.776,A -85,B 0,C 180,E1 -11834.302,E2 -11834.302} C_VEL
LIN {X 0,Y 382.988,Z 221.78,A -85,B 0,C 180,E1 -11837.236,E2 -11837.236} C_VEL
LIN {X 0,Y 382.989,Z 221.776,A -85,B 0,C 180,E1 -11840.42,E2 -11840.42} C_VEL
LIN {X 0,Y 383.012,Z 221.773,A -85,B 0,C 180,E1 -11844.042,E2 -11844.042} C_VEL
LIN {X 0,Y 383.004,Z 221.776,A -85,B 0,C 180,E1 -11846.599,E2 -11846.599} C_VEL
LIN {X 0,Y 382.979,Z 221.778,A -85,B 0,C 180,E1 -11850.299,E2 -11850.299} C_VEL
LIN {X 0,Y 383.008,Z 221.774,A -85,B 0,C 180,E1 -11854.045,E2 -11854.045} C_VEL
LIN {X 0,Y 383.056,Z 221.78,A -85,B 0,C 180,E1 -11857.056,E2 -11857.056} C_VEL
LIN {X 0,Y 384.477,Z 229.541,A -85,B 0,C 180,E1 -11859.16,E2 -11859.16} C_VEL
LIN {X 0,Y 388.681,Z 251.511,A -85,B 0,C 180,E1 -11859.873,E2 -11859.873} C_VEL
LIN {X 0,Y 386.682,Z 337.759,A -85,B 0,C 180,E1 -11861.934,E2 -11861.934} C_VEL
LIN {X 0,Y 386.256,Z 351.234,A -85,B 0,C 180,E1 -11862.46,E2 -11862.46} C_VEL
LIN {X 0,Y 385.798,Z 364.231,A -85,B 0,C 180,E1 -11863.19,E2 -11863.19} C_VEL
LIN {X 0,Y 385.092,Z 376.614,A -85,B 0,C 180,E1 -11864.112,E2 -11864.112} C_VEL
LIN {X 0,Y 384.502,Z 387.839,A -85,B 0,C 180,E1 -11865.173,E2 -11865.173} C_VEL
LIN {X 0,Y 383.899,Z 399.003,A -85,B 0,C 180,E1 -11866.502,E2 -11866.502} C_VEL
LIN {X 0,Y 383.307,Z 408.086,A -85,B 0,C 180,E1 -11867.827,E2 -11867.827} C_VEL
LIN {X 0,Y 382.741,Z 416.885,A -85,B 0,C 180,E1 -11869.419,E2 -11869.419} C_VEL
LIN {X 0,Y 382.335,Z 423.946,A -85,B 0,C 180,E1 -11871.011,E2 -11871.011} C_VEL
LIN {X 0,Y 382.063,Z 429.575,A -85,B 0,C 180,E1 -11872.602,E2 -11872.602} C_VEL
LIN {X 0,Y 381.905,Z 433.942,A -85,B 0,C 180,E1 -11874.191,E2 -11874.191} C_VEL
LIN {X 0,Y 381.771,Z 437.173,A -85,B 0,C 180,E1 -11875.777,E2 -11875.777} C_VEL
LIN {X 0,Y 381.75,Z 438.728,A -85,B 0,C 180,E1 -11876.834,E2 -11876.834} C_VEL
LIN {X 0,Y 381.755,Z 439.847,A -85,B 0,C 180,E1 -11877.89,E2 -11877.89} C_VEL
LIN {X 0,Y 381.711,Z 440.554,A -85,B 0,C 180,E1 -11878.945,E2 -11878.945} C_VEL
LIN {X 0,Y 381.713,Z 440.816,A -85,B 0,C 180,E1 -11880,E2 -11880} C_VEL
LIN {X 0,Y 381.771,Z 440.624,A -85,B 0,C 180,E1 -11881.055,E2 -11881.055} C_VEL
LIN {X 0,Y 381.881,Z 440.021,A -85,B 0,C 180,E1 -11882.109,E2 -11882.109} C_VEL
LIN {X 0,Y 382.076,Z 438.998,A -85,B 0,C 180,E1 -11883.163,E2 -11883.163} C_VEL
LIN {X 0,Y 382.29,Z 437.493,A -85,B 0,C 180,E1 -11884.217,E2 -11884.217} C_VEL
LIN {X 0,Y 382.521,Z 434.429,A -85,B 0,C 180,E1 -11885.799,E2 -11885.799} C_VEL
LIN {X 0,Y 382.979,Z 430.255,A -85,B 0,C 180,E1 -11887.38,E2 -11887.38} C_VEL
LIN {X 0,Y 383.749,Z 423.85,A -85,B 0,C 180,E1 -11889.221,E2 -11889.221} C_VEL
LIN {X 0,Y 384.515,Z 416.841,A -85,B 0,C 180,E1 -11890.798,E2 -11890.798} C_VEL
LIN {X 0,Y 385.483,Z 408.062,A -85,B 0,C 180,E1 -11892.37,E2 -11892.37} C_VEL
LIN {X 0,Y 386.557,Z 398.12,A -85,B 0,C 180,E1 -11893.805,E2 -11893.805} C_VEL
LIN {X 0,Y 387.779,Z 386.757,A -85,B 0,C 180,E1 -11895.101,E2 -11895.101} C_VEL
LIN {X 0,Y 388.844,Z 375.152,A -85,B 0,C 180,E1 -11896.157,E2 -11896.157} C_VEL
LIN {X 0,Y 389.752,Z 363.135,A -85,B 0,C 180,E1 -11897.012,E2 -11897.012} C_VEL
LIN {X 0,Y 390.447,Z 351.377,A -85,B 0,C 180,E1 -11897.654,E2 -11897.654} C_VEL
LIN {X 0,Y 391.075,Z 338.216,A -85,B 0,C 180,E1 -11898.161,E2 -11898.161} C_VEL
LIN {X 0,Y 394.796,Z 255.668,A -85,B 0,C 180,E1 -11900.415,E2 -11900.415} C_VEL
LIN {X 0,Y 393.181,Z 249.517,A -85,B 0,C 180,E1 -11900.773,E2 -11900.773} C_VEL
LIN {X 0,Y 389.195,Z 240.883,A -85,B 0,C 180,E1 -11901.473,E2 -11901.473} C_VEL
LIN {X 0,Y 386.272,Z 235.101,A -85,B 0,C 180,E1 -11901.996,E2 -11901.996} C_VEL
LIN {X 0,Y 384.705,Z 227.929,A -85,B 0,C 180,E1 -11904.846,E2 -11904.846} C_VEL
LIN {X 0,Y 383.067,Z 221.77,A -85,B 0,C 180,E1 -11907.742,E2 -11907.742} C_VEL
LIN {X 0,Y 382.988,Z 221.779,A -85,B 0,C 180,E1 -11910.918,E2 -11910.918} C_VEL
LIN {X 0,Y 383.023,Z 221.774,A -85,B 0,C 180,E1 -11914.667,E2 -11914.667} C_VEL
LIN {X 0,Y 383.004,Z 221.776,A -85,B 0,C 180,E1 -11917.903,E2 -11917.903} C_VEL
LIN {X 0,Y 382.989,Z 221.778,A -85,B 0,C 180,E1 -11921.347,E2 -11921.347} C_VEL
LIN {X 0,Y 383,Z 221.778,A -85,B 0,C 180,E1 -11924.303,E2 -11924.303} C_VEL
LIN {X 0,Y 383.015,Z 221.775,A -85,B 0,C 180,E1 -11927.239,E2 -11927.239} C_VEL
LIN {X 0,Y 383.014,Z 221.777,A -85,B 0,C 180,E1 -11930.414,E2 -11930.414} C_VEL
LIN {X 0,Y 383.029,Z 221.776,A -85,B 0,C 180,E1 -11934.044,E2 -11934.044} C_VEL
LIN {X 0,Y 383.015,Z 221.777,A -85,B 0,C 180,E1 -11935.541,E2 -11935.541} C_VEL
LIN {X 0,Y 384.701,Z 227.858,A -85,B 0,C 180,E1 -11938.007,E2 -11938.007} C_VEL
LIN {X 0,Y 386.734,Z 235.332,A -85,B 0,C 180,E1 -11940.615,E2 -11940.615} C_VEL
LIN {X 0,Y 388.384,Z 243.495,A -85,B 0,C 180,E1 -11943.102,E2 -11943.102} C_VEL
LIN {X 0,Y 388.894,Z 246.723,A -85,B 0,C 180,E1 -11944.007,E2 -11944.007} C_VEL
LIN {X 0,Y 387.037,Z 259.827,A -85,B 0,C 180,E1 -11947.098,E2 -11947.098} C_VEL
LIN {X 0,Y 390.79,Z 276.64,A -85,B 0,C 180,E1 -11948.043,E2 -11948.043} C_VEL
LIN {X 0,Y 393.118,Z 292.144,A -85,B 0,C 180,E1 -11948.759,E2 -11948.759} C_VEL
LIN {X 0,Y 393.393,Z 297.947,A -85,B 0,C 180,E1 -11948.968,E2 -11948.968} C_VEL
LIN {X 0,Y 390.285,Z 372.298,A -85,B 0,C 180,E1 -11950.984,E2 -11950.984} C_VEL
LIN {X 0,Y 389.419,Z 385.296,A -85,B 0,C 180,E1 -11951.52,E2 -11951.52} C_VEL
LIN {X 0,Y 388.388,Z 397.542,A -85,B 0,C 180,E1 -11952.219,E2 -11952.219} C_VEL
LIN {X 0,Y 387.254,Z 409.654,A -85,B 0,C 180,E1 -11953.119,E2 -11953.119} C_VEL
LIN {X 0,Y 386.156,Z 420.744,A -85,B 0,C 180,E1 -11954.156,E2 -11954.156} C_VEL
LIN {X 0,Y 384.931,Z 431.73,A -85,B 0,C 180,E1 -11955.435,E2 -11955.435} C_VEL
LIN {X 0,Y 384.063,Z 441.068,A -85,B 0,C 180,E1 -11956.776,E2 -11956.776} C_VEL
LIN {X 0,Y 383.24,Z 448.689,A -85,B 0,C 180,E1 -11958.093,E2 -11958.093} C_VEL
LIN {X 0,Y 382.554,Z 456.24,A -85,B 0,C 180,E1 -11959.68,E2 -11959.68} C_VEL
LIN {X 0,Y 382.048,Z 463.145,A -85,B 0,C 180,E1 -11961.536,E2 -11961.536} C_VEL
LIN {X 0,Y 381.749,Z 467.739,A -85,B 0,C 180,E1 -11963.126,E2 -11963.126} C_VEL
LIN {X 0,Y 381.63,Z 471.203,A -85,B 0,C 180,E1 -11964.716,E2 -11964.716} C_VEL
LIN {X 0,Y 381.627,Z 472.947,A -85,B 0,C 180,E1 -11965.774,E2 -11965.774} C_VEL
LIN {X 0,Y 381.578,Z 474.206,A -85,B 0,C 180,E1 -11966.831,E2 -11966.831} C_VEL
LIN {X 0,Y 381.653,Z 475.026,A -85,B 0,C 180,E1 -11967.888,E2 -11967.888} C_VEL
LIN {X 0,Y 381.692,Z 475.424,A -85,B 0,C 180,E1 -11968.944,E2 -11968.944} C_VEL
LIN {X 0,Y 381.687,Z 475.383,A -85,B 0,C 180,E1 -11969.999,E2 -11969.999} C_VEL
LIN {X 0,Y 381.694,Z 474.86,A -85,B 0,C 180,E1 -11971.054,E2 -11971.054} C_VEL
LIN {X 0,Y 381.748,Z 473.912,A -85,B 0,C 180,E1 -11972.109,E2 -11972.109} C_VEL
LIN {X 0,Y 381.651,Z 471.331,A -85,B 0,C 180,E1 -11974.223,E2 -11974.223} C_VEL
LIN {X 0,Y 381.697,Z 467.986,A -85,B 0,C 180,E1 -11976.133,E2 -11976.133} C_VEL
LIN {X 0,Y 381.908,Z 463.466,A -85,B 0,C 180,E1 -11977.932,E2 -11977.932} C_VEL
LIN {X 0,Y 382.332,Z 457.202,A -85,B 0,C 180,E1 -11979.789,E2 -11979.789} C_VEL
LIN {X 0,Y 382.923,Z 450.392,A -85,B 0,C 180,E1 -11981.378,E2 -11981.378} C_VEL
LIN {X 0,Y 383.838,Z 441.908,A -85,B 0,C 180,E1 -11982.96,E2 -11982.96} C_VEL
LIN {X 0,Y 384.628,Z 432.913,A -85,B 0,C 180,E1 -11984.317,E2 -11984.317} C_VEL
LIN {X 0,Y 385.786,Z 422.45,A -85,B 0,C 180,E1 -11985.586,E2 -11985.586} C_VEL
LIN {X 0,Y 386.853,Z 411.661,A -85,B 0,C 180,E1 -11986.625,E2 -11986.625} C_VEL
LIN {X 0,Y 387.902,Z 399.568,A -85,B 0,C 180,E1 -11987.529,E2 -11987.529} C_VEL
LIN {X 0,Y 388.821,Z 386.879,A -85,B 0,C 180,E1 -11988.234,E2 -11988.234} C_VEL
LIN {X 0,Y 389.607,Z 374.072,A -85,B 0,C 180,E1 -11988.707,E2 -11988.707} C_VEL
LIN {X 0,Y 389.959,Z 355.004,A -85,B 0,C 180,E1 -11989.123,E2 -11989.123} C_VEL
LIN {X 0,Y 390.806,Z 295.131,A -85,B 0,C 180,E1 -11990.259,E2 -11990.259} C_VEL
LIN {X 0,Y 387.725,Z 273.265,A -85,B 0,C 180,E1 -11990.895,E2 -11990.895} C_VEL
LIN {X 0,Y 384.934,Z 257.235,A -85,B 0,C 180,E1 -11991.416,E2 -11991.416} C_VEL
LIN {X 0,Y 386.392,Z 239.941,A -85,B 0,C 180,E1 -11995.016,E2 -11995.016} C_VEL
LIN {X 0,Y 385.6,Z 234.233,A -85,B 0,C 180,E1 -11996.276,E2 -11996.276} C_VEL
LIN {X 0,Y 383.079,Z 221.769,A -85,B 0,C 180,E1 -11999.162,E2 -11999.162} C_VEL
LIN {X 0,Y 382.983,Z 221.761,A -85,B 0,C 180,E1 -12002.421,E2 -12002.421} C_VEL
LIN {X 0,Y 383.02,Z 221.77,A -85,B 0,C 180,E1 -12005.954,E2 -12005.954} C_VEL
LIN {X 0,Y 382.98,Z 221.772,A -85,B 0,C 180,E1 -12009.58,E2 -12009.58} C_VEL
LIN {X 0,Y 382.999,Z 221.77,A -85,B 0,C 180,E1 -12012.778,E2 -12012.778} C_VEL
LIN {X 0,Y 382.989,Z 221.779,A -85,B 0,C 180,E1 -12015.788,E2 -12015.788} C_VEL
LIN {X 0,Y 382.954,Z 221.768,A -85,B 0,C 180,E1 -12018.8,E2 -12018.8} C_VEL
LIN {X 0,Y 382.986,Z 221.773,A -85,B 0,C 180,E1 -12022.097,E2 -12022.097} C_VEL
LIN {X 0,Y 383.01,Z 221.763,A -85,B 0,C 180,E1 -12025.331,E2 -12025.331} C_VEL
LIN {X 0,Y 382.974,Z 221.769,A -85,B 0,C 180,E1 -12029.081,E2 -12029.081} C_VEL
LIN {X 0,Y 382.961,Z 221.77,A -85,B 0,C 180,E1 -12032.691,E2 -12032.691} C_VEL
LIN {X 0,Y 382.998,Z 221.766,A -85,B 0,C 180,E1 -12036.19,E2 -12036.19} C_VEL
LIN {X 0,Y 383.047,Z 221.76,A -85,B 0,C 180,E1 -12039.598,E2 -12039.598} C_VEL
LIN {X 0,Y 383.084,Z 221.762,A -85,B 0,C 180,E1 -12042.931,E2 -12042.931} C_VEL
LIN {X 0,Y 383.117,Z 221.738,A -85,B 0,C 180,E1 -12046.464,E2 -12046.464} C_VEL
LIN {X 0,Y 383.133,Z 221.763,A -85,B 0,C 180,E1 -12050.498,E2 -12050.498} C_VEL
LIN {X 0,Y 383.22,Z 221.732,A -85,B 0,C 180,E1 -12053.683,E2 -12053.683} C_VEL
LIN {X 0,Y 383.37,Z 221.725,A -85,B 0,C 180,E1 -12057.899,E2 -12057.899} C_VEL
LIN {X 0,Y 383.366,Z 221.709,A -85,B 0,C 180,E1 -12062.101,E2 -12062.101} C_VEL
LIN {X 0,Y 383.25,Z 221.741,A -85,B 0,C 180,E1 -12066.63,E2 -12066.63} C_VEL
LIN {X 0,Y 383.142,Z 221.742,A -85,B 0,C 180,E1 -12069.503,E2 -12069.503} C_VEL
LIN {X 0,Y 383.117,Z 221.758,A -85,B 0,C 180,E1 -12073.537,E2 -12073.537} C_VEL
LIN {X 0,Y 383.086,Z 221.749,A -85,B 0,C 180,E1 -12077.07,E2 -12077.07} C_VEL
LIN {X 0,Y 383.024,Z 221.771,A -85,B 0,C 180,E1 -12080.649,E2 -12080.649} C_VEL
LIN {X 0,Y 383.027,Z 221.76,A -85,B 0,C 180,E1 -12083.808,E2 -12083.808} C_VEL
LIN {X 0,Y 383.05,Z 221.772,A -85,B 0,C 180,E1 -12087.303,E2 -12087.303} C_VEL
LIN {X 0,Y 382.977,Z 221.777,A -85,B 0,C 180,E1 -12090.92,E2 -12090.92} C_VEL
LIN {X 0,Y 383.013,Z 221.767,A -85,B 0,C 180,E1 -12094.669,E2 -12094.669} C_VEL
LIN {X 0,Y 382.997,Z 221.771,A -85,B 0,C 180,E1 -12097.905,E2 -12097.905} C_VEL
LIN {X 0,Y 382.981,Z 221.776,A -85,B 0,C 180,E1 -12101.348,E2 -12101.348} C_VEL
LIN {X 0,Y 382.995,Z 221.778,A -85,B 0,C 180,E1 -12104.305,E2 -12104.305} C_VEL
LIN {X 0,Y 383.007,Z 221.773,A -85,B 0,C 180,E1 -12107.242,E2 -12107.242} C_VEL
LIN {X 0,Y 383.013,Z 221.774,A -85,B 0,C 180,E1 -12110.415,E2 -12110.415} C_VEL
LIN {X 0,Y 383.008,Z 221.778,A -85,B 0,C 180,E1 -12113.987,E2 -12113.987} C_VEL
LIN {X 0,Y 383.818,Z 224.242,A -85,B 0,C 180,E1 -12114.259,E2 -12114.259} C_VEL
LIN {X 0,Y 389.996,Z 238.873,A -85,B 0,C 180,E1 -12114.985,E2 -12114.985} C_VEL
LIN {X 0,Y 392.182,Z 251.475,A -85,B 0,C 180,E1 -12115.382,E2 -12115.382} C_VEL
LIN {X 0,Y 390.623,Z 336.775,A -85,B 0,C 180,E1 -12116.99,E2 -12116.99} C_VEL
LIN {X 0,Y 390.151,Z 349.979,A -85,B 0,C 180,E1 -12117.433,E2 -12117.433} C_VEL
LIN {X 0,Y 389.573,Z 361.619,A -85,B 0,C 180,E1 -12118.024,E2 -12118.024} C_VEL
LIN {X 0,Y 388.703,Z 373.498,A -85,B 0,C 180,E1 -12118.833,E2 -12118.833} C_VEL
LIN {X 0,Y 387.77,Z 384.568,A -85,B 0,C 180,E1 -12119.806,E2 -12119.806} C_VEL
LIN {X 0,Y 386.779,Z 393.977,A -85,B 0,C 180,E1 -12120.831,E2 -12120.831} C_VEL
LIN {X 0,Y 385.822,Z 402.945,A -85,B 0,C 180,E1 -12122.029,E2 -12122.029} C_VEL
LIN {X 0,Y 384.848,Z 411.788,A -85,B 0,C 180,E1 -12123.487,E2 -12123.487} C_VEL
LIN {X 0,Y 383.903,Z 419.692,A -85,B 0,C 180,E1 -12125.1,E2 -12125.1} C_VEL
LIN {X 0,Y 383.271,Z 425.115,A -85,B 0,C 180,E1 -12126.471,E2 -12126.471} C_VEL
LIN {X 0,Y 382.751,Z 429.703,A -85,B 0,C 180,E1 -12127.889,E2 -12127.889} C_VEL
LIN {X 0,Y 382.268,Z 434.164,A -85,B 0,C 180,E1 -12129.66,E2 -12129.66} C_VEL
LIN {X 0,Y 382.039,Z 436.108,A -85,B 0,C 180,E1 -12130.664,E2 -12130.664} C_VEL
LIN {X 0,Y 381.804,Z 437.782,A -85,B 0,C 180,E1 -12131.766,E2 -12131.766} C_VEL
LIN {X 0,Y 381.689,Z 439.338,A -85,B 0,C 180,E1 -12133.232,E2 -12133.232} C_VEL
LIN {X 0,Y 381.533,Z 440.195,A -85,B 0,C 180,E1 -12135.057,E2 -12135.057} C_VEL
LIN {X 0,Y 381.526,Z 440.155,A -85,B 0,C 180,E1 -12136.146,E2 -12136.146} C_VEL
LIN {X 0,Y 381.615,Z 439.546,A -85,B 0,C 180,E1 -12137.444,E2 -12137.444} C_VEL
LIN {X 0,Y 381.654,Z 437.509,A -85,B 0,C 180,E1 -12139.39,E2 -12139.39} C_VEL
LIN {X 0,Y 381.838,Z 434.748,A -85,B 0,C 180,E1 -12141,E2 -12141} C_VEL
LIN {X 0,Y 382.119,Z 430.954,A -85,B 0,C 180,E1 -12142.604,E2 -12142.604} C_VEL
LIN {X 0,Y 382.432,Z 426.041,A -85,B 0,C 180,E1 -12144.2,E2 -12144.2} C_VEL
LIN {X 0,Y 382.907,Z 419.85,A -85,B 0,C 180,E1 -12145.791,E2 -12145.791} C_VEL
LIN {X 0,Y 383.472,Z 412.098,A -85,B 0,C 180,E1 -12147.375,E2 -12147.375} C_VEL
LIN {X 0,Y 384.308,Z 402.45,A -85,B 0,C 180,E1 -12148.953,E2 -12148.953} C_VEL
LIN {X 0,Y 385.116,Z 392.372,A -85,B 0,C 180,E1 -12150.263,E2 -12150.263} C_VEL
LIN {X 0,Y 386.033,Z 381.069,A -85,B 0,C 180,E1 -12151.436,E2 -12151.436} C_VEL
LIN {X 0,Y 386.764,Z 369.9,A -85,B 0,C 180,E1 -12152.345,E2 -12152.345} C_VEL
LIN {X 0,Y 387.31,Z 357.411,A -85,B 0,C 180,E1 -12153.122,E2 -12153.122} C_VEL
LIN {X 0,Y 387.803,Z 344.568,A -85,B 0,C 180,E1 -12153.692,E2 -12153.692} C_VEL
LIN {X 0,Y 388.071,Z 331.445,A -85,B 0,C 180,E1 -12154.052,E2 -12154.052} C_VEL
LIN {X 0,Y 388.39,Z 310.716,A -85,B 0,C 180,E1 -12154.432,E2 -12154.432} C_VEL
LIN {X 0,Y 387.881,Z 304.894,A -85,B 0,C 180,E1 -12154.562,E2 -12154.562} C_VEL
LIN {X 0,Y 382.506,Z 286.171,A -85,B 0,C 180,E1 -12155.144,E2 -12155.144} C_VEL
LIN {X 0,Y 382.034,Z 280.351,A -85,B 0,C 180,E1 -12155.276,E2 -12155.276} C_VEL
LIN {X 0,Y 382.318,Z 250.545,A -85,B 0,C 180,E1 -12155.84,E2 -12155.84} C_VEL
LIN {X 0,Y 379,Z 231.572,A -85,B 0,C 180,E1 -12156.362,E2 -12156.362} C_VEL
LIN {X 0,Y 376.424,Z 223.56,A -85,B 0,C 180,E1 -12156.661,E2 -12156.661} C_VEL
LIN {X 0,Y 376.246,Z 222.62,A -85,B 0,C 180,E1 -12156.773,E2 -12156.773} C_VEL
LIN {X 0,Y 376.119,Z 222.632,A -85,B 0,C 180,E1 -12159.683,E2 -12159.683} C_VEL
LIN {X 0,Y 376.096,Z 222.635,A -85,B 0,C 180,E1 -12163.659,E2 -12163.659} C_VEL
LIN {X 0,Y 376.051,Z 222.641,A -85,B 0,C 180,E1 -12167.608,E2 -12167.608} C_VEL
LIN {X 0,Y 375.985,Z 222.649,A -85,B 0,C 180,E1 -12170.833,E2 -12170.833} C_VEL
LIN {X 0,Y 375.965,Z 222.656,A -85,B 0,C 180,E1 -12174.285,E2 -12174.285} C_VEL
LIN {X 0,Y 375.924,Z 222.66,A -85,B 0,C 180,E1 -12177.866,E2 -12177.866} C_VEL
LIN {X 0,Y 375.963,Z 222.654,A -85,B 0,C 180,E1 -12181.563,E2 -12181.563} C_VEL
LIN {X 0,Y 375.955,Z 222.655,A -85,B 0,C 180,E1 -12185.417,E2 -12185.417} C_VEL
LIN {X 0,Y 375.939,Z 222.655,A -85,B 0,C 180,E1 -12188.263,E2 -12188.263} C_VEL
LIN {X 0,Y 375.919,Z 222.661,A -85,B 0,C 180,E1 -12191.597,E2 -12191.597} C_VEL
LIN {X 0,Y 375.926,Z 222.656,A -85,B 0,C 180,E1 -12194.73,E2 -12194.73} C_VEL
LIN {X 0,Y 375.913,Z 222.66,A -85,B 0,C 180,E1 -12197.696,E2 -12197.696} C_VEL
LIN {X 0,Y 375.938,Z 222.655,A -85,B 0,C 180,E1 -12200.534,E2 -12200.534} C_VEL
LIN {X 0,Y 375.959,Z 222.654,A -85,B 0,C 180,E1 -12203.498,E2 -12203.498} C_VEL
LIN {X 0,Y 375.962,Z 222.651,A -85,B 0,C 180,E1 -12205.888,E2 -12205.888} C_VEL
LIN {X 0,Y 375.965,Z 222.651,A -85,B 0,C 180,E1 -12209.687,E2 -12209.687} C_VEL
LIN {X 0,Y 375.922,Z 222.657,A -85,B 0,C 180,E1 -12212.135,E2 -12212.135} C_VEL
LIN {X 0,Y 375.942,Z 222.658,A -85,B 0,C 180,E1 -12214.534,E2 -12214.534} C_VEL
LIN {X 0,Y 376.042,Z 222.844,A -85,B 0,C 180,E1 -12216.964,E2 -12216.964} C_VEL
LIN {X 0,Y 377.391,Z 230.095,A -85,B 0,C 180,E1 -12218.91,E2 -12218.91} C_VEL
LIN {X 0,Y 380.628,Z 245.947,A -85,B 0,C 180,E1 -12219.437,E2 -12219.437} C_VEL
LIN {X 0,Y 381.736,Z 253.09,A -85,B 0,C 180,E1 -12219.659,E2 -12219.659} C_VEL
LIN {X 0,Y 379.673,Z 338.4,A -85,B 0,C 180,E1 -12221.763,E2 -12221.763} C_VEL
LIN {X 0,Y 379.243,Z 352.445,A -85,B 0,C 180,E1 -12222.334,E2 -12222.334} C_VEL
LIN {X 0,Y 378.809,Z 364.147,A -85,B 0,C 180,E1 -12223.009,E2 -12223.009} C_VEL
LIN {X 0,Y 378.084,Z 376.599,A -85,B 0,C 180,E1 -12223.948,E2 -12223.948} C_VEL
LIN {X 0,Y 377.481,Z 387.978,A -85,B 0,C 180,E1 -12225.037,E2 -12225.037} C_VEL
LIN {X 0,Y 376.927,Z 398.119,A -85,B 0,C 180,E1 -12226.247,E2 -12226.247} C_VEL
LIN {X 0,Y 376.328,Z 407.41,A -85,B 0,C 180,E1 -12227.598,E2 -12227.598} C_VEL
LIN {X 0,Y 375.783,Z 415.078,A -85,B 0,C 180,E1 -12228.948,E2 -12228.948} C_VEL
LIN {X 0,Y 375.354,Z 422.601,A -85,B 0,C 180,E1 -12230.57,E2 -12230.57} C_VEL
LIN {X 0,Y 374.995,Z 429.425,A -85,B 0,C 180,E1 -12232.461,E2 -12232.461} C_VEL
LIN {X 0,Y 374.822,Z 433.532,A -85,B 0,C 180,E1 -12233.928,E2 -12233.928} C_VEL
LIN {X 0,Y 374.7,Z 437.251,A -85,B 0,C 180,E1 -12235.697,E2 -12235.697} C_VEL
LIN {X 0,Y 374.654,Z 438.907,A -85,B 0,C 180,E1 -12236.774,E2 -12236.774} C_VEL
LIN {X 0,Y 374.658,Z 440.076,A -85,B 0,C 180,E1 -12237.85,E2 -12237.85} C_VEL
LIN {X 0,Y 374.645,Z 440.834,A -85,B 0,C 180,E1 -12238.925,E2 -12238.925} C_VEL
LIN {X 0,Y 374.643,Z 441.177,A -85,B 0,C 180,E1 -12240,E2 -12240} C_VEL
LIN {X 0,Y 374.702,Z 441.049,A -85,B 0,C 180,E1 -12241.074,E2 -12241.074} C_VEL
LIN {X 0,Y 374.82,Z 440.495,A -85,B 0,C 180,E1 -12242.149,E2 -12242.149} C_VEL
LIN {X 0,Y 375.024,Z 439.526,A -85,B 0,C 180,E1 -12243.223,E2 -12243.223} C_VEL
LIN {X 0,Y 375.253,Z 438.111,A -85,B 0,C 180,E1 -12244.296,E2 -12244.296} C_VEL
LIN {X 0,Y 375.495,Z 435.144,A -85,B 0,C 180,E1 -12245.908,E2 -12245.908} C_VEL
LIN {X 0,Y 375.987,Z 431.078,A -85,B 0,C 180,E1 -12247.518,E2 -12247.518} C_VEL
LIN {X 0,Y 376.811,Z 424.789,A -85,B 0,C 180,E1 -12249.392,E2 -12249.392} C_VEL
LIN {X 0,Y 377.628,Z 417.944,A -85,B 0,C 180,E1 -12250.997,E2 -12250.997} C_VEL
LIN {X 0,Y 378.682,Z 409.354,A -85,B 0,C 180,E1 -12252.596,E2 -12252.596} C_VEL
LIN {X 0,Y 379.696,Z 400.586,A -85,B 0,C 180,E1 -12253.923,E2 -12253.923} C_VEL
LIN {X 0,Y 380.959,Z 389.84,A -85,B 0,C 180,E1 -12255.241,E2 -12255.241} C_VEL
LIN {X 0,Y 382.185,Z 377.977,A -85,B 0,C 180,E1 -12256.391,E2 -12256.391} C_VEL
LIN {X 0,Y 383.064,Z 367.251,A -85,B 0,C 180,E1 -12257.228,E2 -12257.228} C_VEL
LIN {X 0,Y 383.969,Z 354.466,A -85,B 0,C 180,E1 -12257.992,E2 -12257.992} C_VEL
LIN {X 0,Y 384.703,Z 341.638,A -85,B 0,C 180,E1 -12258.541,E2 -12258.541} C_VEL
LIN {X 0,Y 385.69,Z 318.088,A -85,B 0,C 180,E1 -12259.216,E2 -12259.216} C_VEL
LIN {X 0,Y 388.738,Z 256.614,A -85,B 0,C 180,E1 -12260.969,E2 -12260.969} C_VEL
LIN {X 0,Y 386.714,Z 250.515,A -85,B 0,C 180,E1 -12261.391,E2 -12261.391} C_VEL
LIN {X 0,Y 382.021,Z 241.108,A -85,B 0,C 180,E1 -12262.25,E2 -12262.25} C_VEL
LIN {X 0,Y 379.249,Z 235.748,A -85,B 0,C 180,E1 -12262.785,E2 -12262.785} C_VEL
LIN {X 0,Y 377.917,Z 229.723,A -85,B 0,C 180,E1 -12265.323,E2 -12265.323} C_VEL
LIN {X 0,Y 376.564,Z 224.535,A -85,B 0,C 180,E1 -12267.813,E2 -12267.813} C_VEL
LIN {X 0,Y 375.958,Z 222.655,A -85,B 0,C 180,E1 -12268.836,E2 -12268.836} C_VEL
LIN {X 0,Y 375.963,Z 222.656,A -85,B 0,C 180,E1 -12271.561,E2 -12271.561} C_VEL
LIN {X 0,Y 375.963,Z 222.655,A -85,B 0,C 180,E1 -12275.415,E2 -12275.415} C_VEL
LIN {X 0,Y 375.979,Z 222.652,A -85,B 0,C 180,E1 -12278.27,E2 -12278.27} C_VEL
LIN {X 0,Y 375.939,Z 222.658,A -85,B 0,C 180,E1 -12281.6,E2 -12281.6} C_VEL
LIN {X 0,Y 375.931,Z 222.657,A -85,B 0,C 180,E1 -12285.268,E2 -12285.268} C_VEL
LIN {X 0,Y 375.937,Z 222.656,A -85,B 0,C 180,E1 -12288.399,E2 -12288.399} C_VEL
LIN {X 0,Y 375.975,Z 222.654,A -85,B 0,C 180,E1 -12291.73,E2 -12291.73} C_VEL
LIN {X 0,Y 375.975,Z 222.752,A -85,B 0,C 180,E1 -12294.421,E2 -12294.421} C_VEL
LIN {X 0,Y 377.943,Z 229.39,A -85,B 0,C 180,E1 -12297.365,E2 -12297.365} C_VEL
LIN {X 0,Y 380.06,Z 237.498,A -85,B 0,C 180,E1 -12300.356,E2 -12300.356} C_VEL
LIN {X 0,Y 381.693,Z 245.545,A -85,B 0,C 180,E1 -12302.888,E2 -12302.888} C_VEL
LIN {X 0,Y 382.208,Z 248.737,A -85,B 0,C 180,E1 -12303.811,E2 -12303.811} C_VEL
LIN {X 0,Y 380.589,Z 259.313,A -85,B 0,C 180,E1 -12306.387,E2 -12306.387} C_VEL
LIN {X 0,Y 384.701,Z 277.59,A -85,B 0,C 180,E1 -12307.483,E2 -12307.483} C_VEL
LIN {X 0,Y 386.831,Z 291.824,A -85,B 0,C 180,E1 -12308.177,E2 -12308.177} C_VEL
LIN {X 0,Y 387.294,Z 298.444,A -85,B 0,C 180,E1 -12308.442,E2 -12308.442} C_VEL
LIN {X 0,Y 383.934,Z 372.32,A -85,B 0,C 180,E1 -12310.518,E2 -12310.518} C_VEL
LIN {X 0,Y 382.986,Z 385.082,A -85,B 0,C 180,E1 -12311.059,E2 -12311.059} C_VEL
LIN {X 0,Y 381.725,Z 399.095,A -85,B 0,C 180,E1 -12311.898,E2 -12311.898} C_VEL
LIN {X 0,Y 380.557,Z 410.788,A -85,B 0,C 180,E1 -12312.812,E2 -12312.812} C_VEL
LIN {X 0,Y 379.254,Z 422.683,A -85,B 0,C 180,E1 -12313.998,E2 -12313.998} C_VEL
LIN {X 0,Y 377.92,Z 433.52,A -85,B 0,C 180,E1 -12315.33,E2 -12315.33} C_VEL
LIN {X 0,Y 377.014,Z 443.027,A -85,B 0,C 180,E1 -12316.799,E2 -12316.799} C_VEL
LIN {X 0,Y 375.975,Z 451.567,A -85,B 0,C 180,E1 -12318.407,E2 -12318.407} C_VEL
LIN {X 0,Y 375.378,Z 458.478,A -85,B 0,C 180,E1 -12320.026,E2 -12320.026} C_VEL
LIN {X 0,Y 374.872,Z 464.772,A -85,B 0,C 180,E1 -12321.916,E2 -12321.916} C_VEL
LIN {X 0,Y 374.625,Z 468.898,A -85,B 0,C 180,E1 -12323.536,E2 -12323.536} C_VEL
LIN {X 0,Y 374.54,Z 471.044,A -85,B 0,C 180,E1 -12324.615,E2 -12324.615} C_VEL
LIN {X 0,Y 374.552,Z 472.738,A -85,B 0,C 180,E1 -12325.694,E2 -12325.694} C_VEL
LIN {X 0,Y 374.49,Z 473.941,A -85,B 0,C 180,E1 -12326.771,E2 -12326.771} C_VEL
LIN {X 0,Y 374.552,Z 474.726,A -85,B 0,C 180,E1 -12327.848,E2 -12327.848} C_VEL
LIN {X 0,Y 374.624,Z 475.091,A -85,B 0,C 180,E1 -12328.924,E2 -12328.924} C_VEL
LIN {X 0,Y 374.618,Z 474.979,A -85,B 0,C 180,E1 -12329.999,E2 -12329.999} C_VEL
LIN {X 0,Y 374.628,Z 474.417,A -85,B 0,C 180,E1 -12331.074,E2 -12331.074} C_VEL
LIN {X 0,Y 374.549,Z 472.349,A -85,B 0,C 180,E1 -12333.226,E2 -12333.226} C_VEL
LIN {X 0,Y 374.575,Z 471.096,A -85,B 0,C 180,E1 -12334.303,E2 -12334.303} C_VEL
LIN {X 0,Y 374.593,Z 468.12,A -85,B 0,C 180,E1 -12336.082,E2 -12336.082} C_VEL
LIN {X 0,Y 374.849,Z 463.323,A -85,B 0,C 180,E1 -12338.082,E2 -12338.082} C_VEL
LIN {X 0,Y 375.289,Z 457.109,A -85,B 0,C 180,E1 -12339.974,E2 -12339.974} C_VEL
LIN {X 0,Y 375.924,Z 450.349,A -85,B 0,C 180,E1 -12341.593,E2 -12341.593} C_VEL
LIN {X 0,Y 376.919,Z 441.959,A -85,B 0,C 180,E1 -12343.202,E2 -12343.202} C_VEL
LIN {X 0,Y 377.886,Z 431.937,A -85,B 0,C 180,E1 -12344.736,E2 -12344.736} C_VEL
LIN {X 0,Y 379.086,Z 421.511,A -85,B 0,C 180,E1 -12346.007,E2 -12346.007} C_VEL
LIN {X 0,Y 380.267,Z 410.538,A -85,B 0,C 180,E1 -12347.06,E2 -12347.06} C_VEL
LIN {X 0,Y 381.356,Z 398.258,A -85,B 0,C 180,E1 -12347.979,E2 -12347.979} C_VEL
LIN {X 0,Y 382.243,Z 386.546,A -85,B 0,C 180,E1 -12348.629,E2 -12348.629} C_VEL
LIN {X 0,Y 383.016,Z 373.749,A -85,B 0,C 180,E1 -12349.111,E2 -12349.111} C_VEL
LIN {X 0,Y 383.411,Z 355.079,A -85,B 0,C 180,E1 -12349.524,E2 -12349.524} C_VEL
LIN {X 0,Y 384.328,Z 296.327,A -85,B 0,C 180,E1 -12350.655,E2 -12350.655} C_VEL
LIN {X 0,Y 381.355,Z 274.9,A -85,B 0,C 180,E1 -12351.292,E2 -12351.292} C_VEL
LIN {X 0,Y 378.048,Z 255.883,A -85,B 0,C 180,E1 -12351.942,E2 -12351.942} C_VEL
LIN {X 0,Y 379.396,Z 240.478,A -85,B 0,C 180,E1 -12355.216,E2 -12355.216} C_VEL
LIN {X 0,Y 377.62,Z 230.528,A -85,B 0,C 180,E1 -12357.486,E2 -12357.486} C_VEL
LIN {X 0,Y 376.018,Z 222.649,A -85,B 0,C 180,E1 -12359.38,E2 -12359.38} C_VEL
LIN {X 0,Y 375.945,Z 222.631,A -85,B 0,C 180,E1 -12362.827,E2 -12362.827} C_VEL
LIN {X 0,Y 375.952,Z 222.643,A -85,B 0,C 180,E1 -12365.414,E2 -12365.414} C_VEL
LIN {X 0,Y 375.93,Z 222.65,A -85,B 0,C 180,E1 -12368.262,E2 -12368.262} C_VEL
LIN {X 0,Y 375.913,Z 222.66,A -85,B 0,C 180,E1 -12371.597,E2 -12371.597} C_VEL
LIN {X 0,Y 375.92,Z 222.655,A -85,B 0,C 180,E1 -12374.73,E2 -12374.73} C_VEL
LIN {X 0,Y 375.918,Z 222.647,A -85,B 0,C 180,E1 -12377.698,E2 -12377.698} C_VEL
LIN {X 0,Y 375.927,Z 222.654,A -85,B 0,C 180,E1 -12380.533,E2 -12380.533} C_VEL
LIN {X 0,Y 375.955,Z 222.638,A -85,B 0,C 180,E1 -12383.495,E2 -12383.495} C_VEL
LIN {X 0,Y 375.952,Z 222.649,A -85,B 0,C 180,E1 -12385.888,E2 -12385.888} C_VEL
LIN {X 0,Y 375.953,Z 222.636,A -85,B 0,C 180,E1 -12389.686,E2 -12389.686} C_VEL
LIN {X 0,Y 375.909,Z 222.646,A -85,B 0,C 180,E1 -12392.134,E2 -12392.134} C_VEL
LIN {X 0,Y 375.958,Z 222.643,A -85,B 0,C 180,E1 -12395.716,E2 -12395.716} C_VEL
LIN {X 0,Y 375.971,Z 222.634,A -85,B 0,C 180,E1 -12399.197,E2 -12399.197} C_VEL
LIN {X 0,Y 376.023,Z 222.646,A -85,B 0,C 180,E1 -12402.6,E2 -12402.6} C_VEL
LIN {X 0,Y 376.081,Z 222.613,A -85,B 0,C 180,E1 -12406.342,E2 -12406.342} C_VEL
LIN {X 0,Y 376.103,Z 222.637,A -85,B 0,C 180,E1 -12410.318,E2 -12410.318} C_VEL
LIN {X 0,Y 376.18,Z 222.61,A -85,B 0,C 180,E1 -12413.564,E2 -12413.564} C_VEL
LIN {X 0,Y 376.335,Z 222.601,A -85,B 0,C 180,E1 -12417.86,E2 -12417.86} C_VEL
LIN {X 0,Y 376.331,Z 222.584,A -85,B 0,C 180,E1 -12422.141,E2 -12422.141} C_VEL
LIN {X 0,Y 376.215,Z 222.617,A -85,B 0,C 180,E1 -12426.619,E2 -12426.619} C_VEL
LIN {X 0,Y 376.11,Z 222.615,A -85,B 0,C 180,E1 -12429.682,E2 -12429.682} C_VEL
LIN {X 0,Y 376.081,Z 222.636,A -85,B 0,C 180,E1 -12433.658,E2 -12433.658} C_VEL
LIN {X 0,Y 376.024,Z 222.627,A -85,B 0,C 180,E1 -12437.401,E2 -12437.401} C_VEL
LIN {X 0,Y 375.971,Z 222.65,A -85,B 0,C 180,E1 -12440.833,E2 -12440.833} C_VEL
LIN {X 0,Y 375.987,Z 222.639,A -85,B 0,C 180,E1 -12444.282,E2 -12444.282} C_VEL
LIN {X 0,Y 376.013,Z 222.646,A -85,B 0,C 180,E1 -12446.653,E2 -12446.653} C_VEL
LIN {X 0,Y 375.958,Z 222.649,A -85,B 0,C 180,E1 -12450.314,E2 -12450.314} C_VEL
LIN {X 0,Y 375.954,Z 222.645,A -85,B 0,C 180,E1 -12454.113,E2 -12454.113} C_VEL
LIN {X 0,Y 375.95,Z 222.658,A -85,B 0,C 180,E1 -12456.742,E2 -12456.742} C_VEL
LIN {X 0,Y 375.985,Z 222.653,A -85,B 0,C 180,E1 -12459.972,E2 -12459.972} C_VEL
LIN {X 0,Y 375.928,Z 222.658,A -85,B 0,C 180,E1 -12463.767,E2 -12463.767} C_VEL
LIN {X 0,Y 375.932,Z 222.657,A -85,B 0,C 180,E1 -12466.812,E2 -12466.812} C_VEL
LIN {X 0,Y 375.961,Z 222.654,A -85,B 0,C 180,E1 -12470.539,E2 -12470.539} C_VEL
LIN {X 0,Y 375.979,Z 222.651,A -85,B 0,C 180,E1 -12473.535,E2 -12473.535} C_VEL
LIN {X 0,Y 376.481,Z 224.528,A -85,B 0,C 180,E1 -12473.728,E2 -12473.728} C_VEL
LIN {X 0,Y 382.86,Z 238.818,A -85,B 0,C 180,E1 -12474.49,E2 -12474.49} C_VEL
LIN {X 0,Y 384.026,Z 242.193,A -85,B 0,C 180,E1 -12474.641,E2 -12474.641} C_VEL
LIN {X 0,Y 385.728,Z 252.187,A -85,B 0,C 180,E1 -12474.962,E2 -12474.962} C_VEL
LIN {X 0,Y 384.085,Z 337.088,A -85,B 0,C 180,E1 -12476.589,E2 -12476.589} C_VEL
LIN {X 0,Y 383.602,Z 349.843,A -85,B 0,C 180,E1 -12477.022,E2 -12477.022} C_VEL
LIN {X 0,Y 382.957,Z 362.064,A -85,B 0,C 180,E1 -12477.648,E2 -12477.648} C_VEL
LIN {X 0,Y 381.986,Z 374.696,A -85,B 0,C 180,E1 -12478.531,E2 -12478.531} C_VEL
LIN {X 0,Y 381.025,Z 385.602,A -85,B 0,C 180,E1 -12479.522,E2 -12479.522} C_VEL
LIN {X 0,Y 379.837,Z 396.289,A -85,B 0,C 180,E1 -12480.747,E2 -12480.747} C_VEL
LIN {X 0,Y 378.768,Z 405.535,A -85,B 0,C 180,E1 -12482.064,E2 -12482.064} C_VEL
LIN {X 0,Y 377.8,Z 413.666,A -85,B 0,C 180,E1 -12483.485,E2 -12483.485} C_VEL
LIN {X 0,Y 376.801,Z 421.479,A -85,B 0,C 180,E1 -12485.188,E2 -12485.188} C_VEL
LIN {X 0,Y 376.051,Z 427.661,A -85,B 0,C 180,E1 -12486.893,E2 -12486.893} C_VEL
LIN {X 0,Y 375.477,Z 432.467,A -85,B 0,C 180,E1 -12488.594,E2 -12488.594} C_VEL
LIN {X 0,Y 375.049,Z 436.056,A -85,B 0,C 180,E1 -12490.289,E2 -12490.289} C_VEL
LIN {X 0,Y 374.805,Z 437.825,A -85,B 0,C 180,E1 -12491.413,E2 -12491.413} C_VEL
LIN {X 0,Y 374.617,Z 439.64,A -85,B 0,C 180,E1 -12493.096,E2 -12493.096} C_VEL
LIN {X 0,Y 374.452,Z 440.484,A -85,B 0,C 180,E1 -12494.767,E2 -12494.767} C_VEL
LIN {X 0,Y 374.433,Z 440.504,A -85,B 0,C 180,E1 -12495.878,E2 -12495.878} C_VEL
LIN {X 0,Y 374.514,Z 439.887,A -85,B 0,C 180,E1 -12497.376,E2 -12497.376} C_VEL
LIN {X 0,Y 374.546,Z 438.099,A -85,B 0,C 180,E1 -12499.186,E2 -12499.186} C_VEL
LIN {X 0,Y 374.736,Z 435.461,A -85,B 0,C 180,E1 -12500.828,E2 -12500.828} C_VEL
LIN {X 0,Y 375.003,Z 431.799,A -85,B 0,C 180,E1 -12502.463,E2 -12502.463} C_VEL
LIN {X 0,Y 375.347,Z 427.021,A -85,B 0,C 180,E1 -12504.09,E2 -12504.09} C_VEL
LIN {X 0,Y 375.785,Z 420.996,A -85,B 0,C 180,E1 -12505.711,E2 -12505.711} C_VEL
LIN {X 0,Y 376.375,Z 413.491,A -85,B 0,C 180,E1 -12507.326,E2 -12507.326} C_VEL
LIN {X 0,Y 377.193,Z 404.056,A -85,B 0,C 180,E1 -12508.934,E2 -12508.934} C_VEL
LIN {X 0,Y 378.038,Z 394.342,A -85,B 0,C 180,E1 -12510.267,E2 -12510.267} C_VEL
LIN {X 0,Y 378.944,Z 383.398,A -85,B 0,C 180,E1 -12511.462,E2 -12511.462} C_VEL
LIN {X 0,Y 379.676,Z 372.778,A -85,B 0,C 180,E1 -12512.388,E2 -12512.388} C_VEL
LIN {X 0,Y 380.279,Z 361.209,A -85,B 0,C 180,E1 -12513.179,E2 -12513.179} C_VEL
LIN {X 0,Y 380.829,Z 347.657,A -85,B 0,C 180,E1 -12513.844,E2 -12513.844} C_VEL
LIN {X 0,Y 381.185,Z 334.676,A -85,B 0,C 180,E1 -12514.256,E2 -12514.256} C_VEL
LIN {X 0,Y 382.034,Z 280.351,A -85,B 0,C 180,E1 -12515.276,E2 -12515.276} C_VEL
LIN {X 0,Y 381.693,Z 274.532,A -85,B 0,C 180,E1 -12515.404,E2 -12515.404} C_VEL
LIN {X 0,Y 379.415,Z 265.117,A -85,B 0,C 180,E1 -12515.687,E2 -12515.687} C_VEL
LIN {X 0,Y 377.082,Z 257.651,A -85,B 0,C 180,E1 -12515.939,E2 -12515.939} C_VEL
LIN {X 0,Y 375.302,Z 250.031,A -85,B 0,C 180,E1 -12516.171,E2 -12516.171} C_VEL
LIN {X 0,Y 372.349,Z 233.412,A -85,B 0,C 180,E1 -12516.64,E2 -12516.64} C_VEL
LIN {X 0,Y 369.242,Z 223.701,A -85,B 0,C 180,E1 -12517.005,E2 -12517.005} C_VEL
LIN {X 0,Y 369.143,Z 223.506,A -85,B 0,C 180,E1 -12517.66,E2 -12517.66} C_VEL
LIN {X 0,Y 369.026,Z 223.517,A -85,B 0,C 180,E1 -12520.98,E2 -12520.98} C_VEL
LIN {X 0,Y 369.021,Z 223.52,A -85,B 0,C 180,E1 -12524.336,E2 -12524.336} C_VEL
LIN {X 0,Y 369.008,Z 223.518,A -85,B 0,C 180,E1 -12527.769,E2 -12527.769} C_VEL
LIN {X 0,Y 368.916,Z 223.529,A -85,B 0,C 180,E1 -12531.222,E2 -12531.222} C_VEL
LIN {X 0,Y 368.925,Z 223.531,A -85,B 0,C 180,E1 -12533.878,E2 -12533.878} C_VEL
LIN {X 0,Y 368.865,Z 223.535,A -85,B 0,C 180,E1 -12537.213,E2 -12537.213} C_VEL
LIN {X 0,Y 368.899,Z 223.534,A -85,B 0,C 180,E1 -12539.693,E2 -12539.693} C_VEL
LIN {X 0,Y 368.902,Z 223.531,A -85,B 0,C 180,E1 -12543.043,E2 -12543.043} C_VEL
LIN {X 0,Y 368.917,Z 223.53,A -85,B 0,C 180,E1 -12546.198,E2 -12546.198} C_VEL
LIN {X 0,Y 368.878,Z 223.534,A -85,B 0,C 180,E1 -12548.958,E2 -12548.958} C_VEL
LIN {X 0,Y 368.864,Z 223.537,A -85,B 0,C 180,E1 -12552.006,E2 -12552.006} C_VEL
LIN {X 0,Y 368.879,Z 223.537,A -85,B 0,C 180,E1 -12555.175,E2 -12555.175} C_VEL
LIN {X 0,Y 368.866,Z 223.535,A -85,B 0,C 180,E1 -12558.175,E2 -12558.175} C_VEL
LIN {X 0,Y 368.879,Z 223.538,A -85,B 0,C 180,E1 -12561.367,E2 -12561.367} C_VEL
LIN {X 0,Y 368.933,Z 223.531,A -85,B 0,C 180,E1 -12565.146,E2 -12565.146} C_VEL
LIN {X 0,Y 368.902,Z 223.535,A -85,B 0,C 180,E1 -12569.043,E2 -12569.043} C_VEL
LIN {X 0,Y 368.912,Z 223.53,A -85,B 0,C 180,E1 -12571.558,E2 -12571.558} C_VEL
LIN {X 0,Y 368.892,Z 223.534,A -85,B 0,C 180,E1 -12575.22,E2 -12575.22} C_VEL
LIN {X 0,Y 368.996,Z 223.62,A -85,B 0,C 180,E1 -12576.795,E2 -12576.795} C_VEL
LIN {X 0,Y 370.155,Z 230.092,A -85,B 0,C 180,E1 -12578.602,E2 -12578.602} C_VEL
LIN {X 0,Y 372.731,Z 241.069,A -85,B 0,C 180,E1 -12579.014,E2 -12579.014} C_VEL
LIN {X 0,Y 374.832,Z 253.869,A -85,B 0,C 180,E1 -12579.427,E2 -12579.427} C_VEL
LIN {X 0,Y 372.685,Z 338.893,A -85,B 0,C 180,E1 -12581.586,E2 -12581.586} C_VEL
LIN {X 0,Y 372.262,Z 352.104,A -85,B 0,C 180,E1 -12582.134,E2 -12582.134} C_VEL
LIN {X 0,Y 371.812,Z 363.978,A -85,B 0,C 180,E1 -12582.821,E2 -12582.821} C_VEL
LIN {X 0,Y 371.086,Z 376.512,A -85,B 0,C 180,E1 -12583.778,E2 -12583.778} C_VEL
LIN {X 0,Y 370.448,Z 388.149,A -85,B 0,C 180,E1 -12584.907,E2 -12584.907} C_VEL
LIN {X 0,Y 369.896,Z 398.181,A -85,B 0,C 180,E1 -12586.121,E2 -12586.121} C_VEL
LIN {X 0,Y 369.203,Z 408.369,A -85,B 0,C 180,E1 -12587.634,E2 -12587.634} C_VEL
LIN {X 0,Y 368.659,Z 415.943,A -85,B 0,C 180,E1 -12589.01,E2 -12589.01} C_VEL
LIN {X 0,Y 368.261,Z 423.345,A -85,B 0,C 180,E1 -12590.664,E2 -12590.664} C_VEL
LIN {X 0,Y 367.927,Z 429.243,A -85,B 0,C 180,E1 -12592.316,E2 -12592.316} C_VEL
LIN {X 0,Y 367.723,Z 433.882,A -85,B 0,C 180,E1 -12593.975,E2 -12593.975} C_VEL
LIN {X 0,Y 367.633,Z 437.314,A -85,B 0,C 180,E1 -12595.614,E2 -12595.614} C_VEL
LIN {X 0,Y 367.562,Z 439.046,A -85,B 0,C 180,E1 -12596.711,E2 -12596.711} C_VEL
LIN {X 0,Y 367.562,Z 440.3,A -85,B 0,C 180,E1 -12597.808,E2 -12597.808} C_VEL
LIN {X 0,Y 367.561,Z 441.11,A -85,B 0,C 180,E1 -12598.904,E2 -12598.904} C_VEL
LIN {X 0,Y 367.575,Z 441.51,A -85,B 0,C 180,E1 -12600,E2 -12600} C_VEL
LIN {X 0,Y 367.635,Z 441.478,A -85,B 0,C 180,E1 -12601.095,E2 -12601.095} C_VEL
LIN {X 0,Y 367.76,Z 440.977,A -85,B 0,C 180,E1 -12602.19,E2 -12602.19} C_VEL
LIN {X 0,Y 367.975,Z 440.061,A -85,B 0,C 180,E1 -12603.284,E2 -12603.284} C_VEL
LIN {X 0,Y 368.219,Z 438.73,A -85,B 0,C 180,E1 -12604.378,E2 -12604.378} C_VEL
LIN {X 0,Y 368.472,Z 435.867,A -85,B 0,C 180,E1 -12606.021,E2 -12606.021} C_VEL
LIN {X 0,Y 369.012,Z 431.919,A -85,B 0,C 180,E1 -12607.661,E2 -12607.661} C_VEL
LIN {X 0,Y 369.877,Z 425.778,A -85,B 0,C 180,E1 -12609.57,E2 -12609.57} C_VEL
LIN {X 0,Y 370.749,Z 419.067,A -85,B 0,C 180,E1 -12611.204,E2 -12611.204} C_VEL
LIN {X 0,Y 371.895,Z 410.716,A -85,B 0,C 180,E1 -12612.829,E2 -12612.829} C_VEL
LIN {X 0,Y 373.203,Z 400.239,A -85,B 0,C 180,E1 -12614.449,E2 -12614.449} C_VEL
LIN {X 0,Y 374.436,Z 390.536,A -85,B 0,C 180,E1 -12615.653,E2 -12615.653} C_VEL
LIN {X 0,Y 375.76,Z 378.438,A -85,B 0,C 180,E1 -12616.852,E2 -12616.852} C_VEL
LIN {X 0,Y 376.781,Z 367.267,A -85,B 0,C 180,E1 -12617.737,E2 -12617.737} C_VEL
LIN {X 0,Y 377.732,Z 354.478,A -85,B 0,C 180,E1 -12618.509,E2 -12618.509} C_VEL
LIN {X 0,Y 378.529,Z 341.65,A -85,B 0,C 180,E1 -12619.066,E2 -12619.066} C_VEL
LIN {X 0,Y 379.625,Z 317.373,A -85,B 0,C 180,E1 -12619.782,E2 -12619.782} C_VEL
LIN {X 0,Y 382.858,Z 258.374,A -85,B 0,C 180,E1 -12621.517,E2 -12621.517} C_VEL
LIN {X 0,Y 380.585,Z 252.361,A -85,B 0,C 180,E1 -12621.989,E2 -12621.989} C_VEL
LIN {X 0,Y 375.445,Z 242.383,A -85,B 0,C 180,E1 -12622.984,E2 -12622.984} C_VEL
LIN {X 0,Y 372.269,Z 236.415,A -85,B 0,C 180,E1 -12623.652,E2 -12623.652} C_VEL
LIN {X 0,Y 371.187,Z 231.564,A -85,B 0,C 180,E1 -12625.816,E2 -12625.816} C_VEL
LIN {X 0,Y 369.792,Z 226.606,A -85,B 0,C 180,E1 -12628.368,E2 -12628.368} C_VEL
LIN {X 0,Y 368.932,Z 223.531,A -85,B 0,C 180,E1 -12630.24,E2 -12630.24} C_VEL
LIN {X 0,Y 368.902,Z 223.533,A -85,B 0,C 180,E1 -12633.537,E2 -12633.537} C_VEL
LIN {X 0,Y 368.907,Z 223.534,A -85,B 0,C 180,E1 -12636.855,E2 -12636.855} C_VEL
LIN {X 0,Y 368.916,Z 223.531,A -85,B 0,C 180,E1 -12640.369,E2 -12640.369} C_VEL
LIN {X 0,Y 368.887,Z 223.535,A -85,B 0,C 180,E1 -12643.615,E2 -12643.615} C_VEL
LIN {X 0,Y 368.89,Z 223.534,A -85,B 0,C 180,E1 -12646.695,E2 -12646.695} C_VEL
LIN {X 0,Y 368.913,Z 223.531,A -85,B 0,C 180,E1 -12649.643,E2 -12649.643} C_VEL
LIN {X 0,Y 368.937,Z 223.732,A -85,B 0,C 180,E1 -12653.137,E2 -12653.137} C_VEL
LIN {X 0,Y 370.668,Z 229.422,A -85,B 0,C 180,E1 -12655.99,E2 -12655.99} C_VEL
LIN {X 0,Y 372.344,Z 235.496,A -85,B 0,C 180,E1 -12658.514,E2 -12658.514} C_VEL
LIN {X 0,Y 373.846,Z 241.623,A -85,B 0,C 180,E1 -12660.738,E2 -12660.738} C_VEL
LIN {X 0,Y 375.341,Z 249.7,A -85,B 0,C 180,E1 -12663.295,E2 -12663.295} C_VEL
LIN {X 0,Y 375.271,Z 252.366,A -85,B 0,C 180,E1 -12664.018,E2 -12664.018} C_VEL
LIN {X 0,Y 374.216,Z 258.805,A -85,B 0,C 180,E1 -12665.626,E2 -12665.626} C_VEL
LIN {X 0,Y 378.385,Z 277.027,A -85,B 0,C 180,E1 -12666.8,E2 -12666.8} C_VEL
LIN {X 0,Y 380.587,Z 290.526,A -85,B 0,C 180,E1 -12667.521,E2 -12667.521} C_VEL
LIN {X 0,Y 381.278,Z 299.028,A -85,B 0,C 180,E1 -12667.89,E2 -12667.89} C_VEL
LIN {X 0,Y 377.669,Z 371.827,A -85,B 0,C 180,E1 -12670.004,E2 -12670.004} C_VEL
LIN {X 0,Y 376.608,Z 385.118,A -85,B 0,C 180,E1 -12670.584,E2 -12670.584} C_VEL
LIN {X 0,Y 375.275,Z 398.929,A -85,B 0,C 180,E1 -12671.435,E2 -12671.435} C_VEL
LIN {X 0,Y 374.016,Z 410.519,A -85,B 0,C 180,E1 -12672.361,E2 -12672.361} C_VEL
LIN {X 0,Y 372.634,Z 422.345,A -85,B 0,C 180,E1 -12673.565,E2 -12673.565} C_VEL
LIN {X 0,Y 371.297,Z 432.786,A -85,B 0,C 180,E1 -12674.871,E2 -12674.871} C_VEL
LIN {X 0,Y 370.264,Z 441.855,A -85,B 0,C 180,E1 -12676.274,E2 -12676.274} C_VEL
LIN {X 0,Y 369.167,Z 450.512,A -85,B 0,C 180,E1 -12677.911,E2 -12677.911} C_VEL
LIN {X 0,Y 368.442,Z 457.534,A -85,B 0,C 180,E1 -12679.558,E2 -12679.558} C_VEL
LIN {X 0,Y 367.959,Z 463.181,A -85,B 0,C 180,E1 -12681.21,E2 -12681.21} C_VEL
LIN {X 0,Y 367.604,Z 467.6,A -85,B 0,C 180,E1 -12682.86,E2 -12682.86} C_VEL
LIN {X 0,Y 367.456,Z 470.905,A -85,B 0,C 180,E1 -12684.511,E2 -12684.511} C_VEL
LIN {X 0,Y 367.456,Z 472.519,A -85,B 0,C 180,E1 -12685.611,E2 -12685.611} C_VEL
LIN {X 0,Y 367.405,Z 473.683,A -85,B 0,C 180,E1 -12686.709,E2 -12686.709} C_VEL
LIN {X 0,Y 367.451,Z 474.43,A -85,B 0,C 180,E1 -12687.807,E2 -12687.807} C_VEL
LIN {X 0,Y 367.556,Z 474.74,A -85,B 0,C 180,E1 -12688.903,E2 -12688.903} C_VEL
LIN {X 0,Y 367.551,Z 474.565,A -85,B 0,C 180,E1 -12689.999,E2 -12689.999} C_VEL
LIN {X 0,Y 367.563,Z 473.962,A -85,B 0,C 180,E1 -12691.094,E2 -12691.094} C_VEL
LIN {X 0,Y 367.46,Z 472.094,A -85,B 0,C 180,E1 -12693.288,E2 -12693.288} C_VEL
LIN {X 0,Y 367.479,Z 470.86,A -85,B 0,C 180,E1 -12694.386,E2 -12694.386} C_VEL
LIN {X 0,Y 367.521,Z 468.165,A -85,B 0,C 180,E1 -12696.076,E2 -12696.076} C_VEL
LIN {X 0,Y 367.684,Z 464.612,A -85,B 0,C 180,E1 -12697.688,E2 -12697.688} C_VEL
LIN {X 0,Y 368.012,Z 459.864,A -85,B 0,C 180,E1 -12699.341,E2 -12699.341} C_VEL
LIN {X 0,Y 368.682,Z 452.742,A -85,B 0,C 180,E1 -12701.266,E2 -12701.266} C_VEL
LIN {X 0,Y 369.626,Z 444.994,A -85,B 0,C 180,E1 -12702.908,E2 -12702.908} C_VEL
LIN {X 0,Y 370.462,Z 437.084,A -85,B 0,C 180,E1 -12704.276,E2 -12704.276} C_VEL
LIN {X 0,Y 371.597,Z 427.433,A -85,B 0,C 180,E1 -12705.634,E2 -12705.634} C_VEL
LIN {X 0,Y 372.872,Z 416.705,A -85,B 0,C 180,E1 -12706.844,E2 -12706.844} C_VEL
LIN {X 0,Y 374.158,Z 404.477,A -85,B 0,C 180,E1 -12707.912,E2 -12707.912} C_VEL
LIN {X 0,Y 375.14,Z 392.518,A -85,B 0,C 180,E1 -12708.712,E2 -12708.712} C_VEL
LIN {X 0,Y 376.096,Z 380.095,A -85,B 0,C 180,E1 -12709.299,E2 -12709.299} C_VEL
LIN {X 0,Y 376.684,Z 366.713,A -85,B 0,C 180,E1 -12709.706,E2 -12709.706} C_VEL
LIN {X 0,Y 377.847,Z 296.985,A -85,B 0,C 180,E1 -12711.079,E2 -12711.079} C_VEL
LIN {X 0,Y 374.991,Z 276.345,A -85,B 0,C 180,E1 -12711.712,E2 -12711.712} C_VEL
LIN {X 0,Y 371.198,Z 254.535,A -85,B 0,C 180,E1 -12712.48,E2 -12712.48} C_VEL
LIN {X 0,Y 372.393,Z 241.453,A -85,B 0,C 180,E1 -12715.312,E2 -12715.312} C_VEL
LIN {X 0,Y 370.555,Z 231.255,A -85,B 0,C 180,E1 -12717.687,E2 -12717.687} C_VEL
LIN {X 0,Y 368.958,Z 223.528,A -85,B 0,C 180,E1 -12719.58,E2 -12719.58} C_VEL
LIN {X 0,Y 368.892,Z 223.505,A -85,B 0,C 180,E1 -12723.537,E2 -12723.537} C_VEL
LIN {X 0,Y 368.894,Z 223.533,A -85,B 0,C 180,E1 -12726.854,E2 -12726.854} C_VEL
LIN {X 0,Y 368.877,Z 223.535,A -85,B 0,C 180,E1 -12730.373,E2 -12730.373} C_VEL
LIN {X 0,Y 368.875,Z 223.527,A -85,B 0,C 180,E1 -12733.615,E2 -12733.615} C_VEL
LIN {X 0,Y 368.878,Z 223.533,A -85,B 0,C 180,E1 -12736.695,E2 -12736.695} C_VEL
LIN {X 0,Y 368.876,Z 223.53,A -85,B 0,C 180,E1 -12739.647,E2 -12739.647} C_VEL
LIN {X 0,Y 368.892,Z 223.521,A -85,B 0,C 180,E1 -12743.144,E2 -12743.144} C_VEL
LIN {X 0,Y 368.889,Z 223.528,A -85,B 0,C 180,E1 -12746.461,E2 -12746.461} C_VEL
LIN {X 0,Y 368.921,Z 223.519,A -85,B 0,C 180,E1 -12749.046,E2 -12749.046} C_VEL
LIN {X 0,Y 368.849,Z 223.528,A -85,B 0,C 180,E1 -12752.788,E2 -12752.788} C_VEL
LIN {X 0,Y 368.91,Z 223.521,A -85,B 0,C 180,E1 -12756.122,E2 -12756.122} C_VEL
LIN {X 0,Y 368.92,Z 223.519,A -85,B 0,C 180,E1 -12759.946,E2 -12759.946} C_VEL
LIN {X 0,Y 368.955,Z 223.518,A -85,B 0,C 180,E1 -12763.398,E2 -12763.398} C_VEL
LIN {X 0,Y 369.049,Z 223.491,A -85,B 0,C 180,E1 -12766.79,E2 -12766.79} C_VEL
LIN {X 0,Y 369.053,Z 223.513,A -85,B 0,C 180,E1 -12770.132,E2 -12770.132} C_VEL
LIN {X 0,Y 369.142,Z 223.486,A -85,B 0,C 180,E1 -12773.441,E2 -12773.441} C_VEL
LIN {X 0,Y 369.299,Z 223.477,A -85,B 0,C 180,E1 -12777.819,E2 -12777.819} C_VEL
LIN {X 0,Y 369.23,Z 223.477,A -85,B 0,C 180,E1 -12781.091,E2 -12781.091} C_VEL
LIN {X 0,Y 369.295,Z 223.459,A -85,B 0,C 180,E1 -12782.182,E2 -12782.182} C_VEL
LIN {X 0,Y 369.186,Z 223.493,A -85,B 0,C 180,E1 -12786.604,E2 -12786.604} C_VEL
LIN {X 0,Y 369.058,Z 223.491,A -85,B 0,C 180,E1 -12789.869,E2 -12789.869} C_VEL
LIN {X 0,Y 369.029,Z 223.515,A -85,B 0,C 180,E1 -12793.773,E2 -12793.773} C_VEL
LIN {X 0,Y 368.983,Z 223.505,A -85,B 0,C 180,E1 -12797.744,E2 -12797.744} C_VEL
LIN {X 0,Y 368.923,Z 223.53,A -85,B 0,C 180,E1 -12801.22,E2 -12801.22} C_VEL
LIN {X 0,Y 368.951,Z 223.517,A -85,B 0,C 180,E1 -12804.776,E2 -12804.776} C_VEL
LIN {X 0,Y 368.956,Z 223.528,A -85,B 0,C 180,E1 -12807.204,E2 -12807.204} C_VEL
LIN {X 0,Y 368.923,Z 223.527,A -85,B 0,C 180,E1 -12810.955,E2 -12810.955} C_VEL
LIN {X 0,Y 368.924,Z 223.525,A -85,B 0,C 180,E1 -12815.003,E2 -12815.003} C_VEL
LIN {X 0,Y 368.906,Z 223.526,A -85,B 0,C 180,E1 -12818.642,E2 -12818.642} C_VEL
LIN {X 0,Y 368.877,Z 223.53,A -85,B 0,C 180,E1 -12822.011,E2 -12822.011} C_VEL
LIN {X 0,Y 368.879,Z 223.533,A -85,B 0,C 180,E1 -12825.178,E2 -12825.178} C_VEL
LIN {X 0,Y 368.88,Z 223.534,A -85,B 0,C 180,E1 -12828.179,E2 -12828.179} C_VEL
LIN {X 0,Y 368.906,Z 223.531,A -85,B 0,C 180,E1 -12831.361,E2 -12831.361} C_VEL
LIN {X 0,Y 368.935,Z 223.735,A -85,B 0,C 180,E1 -12833.094,E2 -12833.094} C_VEL
LIN {X 0,Y 370.114,Z 226.656,A -85,B 0,C 180,E1 -12833.286,E2 -12833.286} C_VEL
LIN {X 0,Y 376.911,Z 241.856,A -85,B 0,C 180,E1 -12834.123,E2 -12834.123} C_VEL
LIN {X 0,Y 377.901,Z 245.15,A -85,B 0,C 180,E1 -12834.264,E2 -12834.264} C_VEL
LIN {X 0,Y 379.28,Z 254.25,A -85,B 0,C 180,E1 -12834.552,E2 -12834.552} C_VEL
LIN {X 0,Y 377.562,Z 337.588,A -85,B 0,C 180,E1 -12836.175,E2 -12836.175} C_VEL
LIN {X 0,Y 377.058,Z 350.535,A -85,B 0,C 180,E1 -12836.625,E2 -12836.625} C_VEL
LIN {X 0,Y 376.422,Z 361.971,A -85,B 0,C 180,E1 -12837.219,E2 -12837.219} C_VEL
LIN {X 0,Y 375.437,Z 374.173,A -85,B 0,C 180,E1 -12838.075,E2 -12838.075} C_VEL
LIN {X 0,Y 374.41,Z 385.228,A -85,B 0,C 180,E1 -12839.081,E2 -12839.081} C_VEL
LIN {X 0,Y 373.201,Z 395.74,A -85,B 0,C 180,E1 -12840.282,E2 -12840.282} C_VEL
LIN {X 0,Y 372.116,Z 404.49,A -85,B 0,C 180,E1 -12841.519,E2 -12841.519} C_VEL
LIN {X 0,Y 371.117,Z 412.849,A -85,B 0,C 180,E1 -12842.969,E2 -12842.969} C_VEL
LIN {X 0,Y 369.998,Z 420.937,A -85,B 0,C 180,E1 -12844.7,E2 -12844.7} C_VEL
LIN {X 0,Y 369.197,Z 427.288,A -85,B 0,C 180,E1 -12846.439,E2 -12846.439} C_VEL
LIN {X 0,Y 368.525,Z 432.243,A -85,B 0,C 180,E1 -12848.17,E2 -12848.17} C_VEL
LIN {X 0,Y 368.059,Z 435.972,A -85,B 0,C 180,E1 -12849.899,E2 -12849.899} C_VEL
LIN {X 0,Y 367.788,Z 437.861,A -85,B 0,C 180,E1 -12851.045,E2 -12851.045} C_VEL
LIN {X 0,Y 367.557,Z 439.939,A -85,B 0,C 180,E1 -12852.951,E2 -12852.951} C_VEL
LIN {X 0,Y 367.395,Z 440.759,A -85,B 0,C 180,E1 -12854.467,E2 -12854.467} C_VEL
LIN {X 0,Y 367.333,Z 440.854,A -85,B 0,C 180,E1 -12855.599,E2 -12855.599} C_VEL
LIN {X 0,Y 367.415,Z 440.226,A -85,B 0,C 180,E1 -12857.304,E2 -12857.304} C_VEL
LIN {X 0,Y 367.452,Z 438.683,A -85,B 0,C 180,E1 -12858.975,E2 -12858.975} C_VEL
LIN {X 0,Y 367.545,Z 437.103,A -85,B 0,C 180,E1 -12860.092,E2 -12860.092} C_VEL
LIN {X 0,Y 367.807,Z 433.915,A -85,B 0,C 180,E1 -12861.762,E2 -12861.762} C_VEL
LIN {X 0,Y 368.139,Z 429.659,A -85,B 0,C 180,E1 -12863.424,E2 -12863.424} C_VEL
LIN {X 0,Y 368.458,Z 424.238,A -85,B 0,C 180,E1 -12865.077,E2 -12865.077} C_VEL
LIN {X 0,Y 369.071,Z 417.443,A -85,B 0,C 180,E1 -12866.726,E2 -12866.726} C_VEL
LIN {X 0,Y 369.849,Z 408.915,A -85,B 0,C 180,E1 -12868.368,E2 -12868.368} C_VEL
LIN {X 0,Y 370.581,Z 400.211,A -85,B 0,C 180,E1 -12869.73,E2 -12869.73} C_VEL
LIN {X 0,Y 371.428,Z 390.666,A -85,B 0,C 180,E1 -12870.95,E2 -12870.95} C_VEL
LIN {X 0,Y 372.275,Z 380.172,A -85,B 0,C 180,E1 -12872.03,E2 -12872.03} C_VEL
LIN {X 0,Y 373.088,Z 368.536,A -85,B 0,C 180,E1 -12872.971,E2 -12872.971} C_VEL
LIN {X 0,Y 373.673,Z 356.416,A -85,B 0,C 180,E1 -12873.722,E2 -12873.722} C_VEL
LIN {X 0,Y 374.136,Z 344.076,A -85,B 0,C 180,E1 -12874.261,E2 -12874.261} C_VEL
LIN {X 0,Y 374.401,Z 330.688,A -85,B 0,C 180,E1 -12874.624,E2 -12874.624} C_VEL
LIN {X 0,Y 375.6,Z 252.035,A -85,B 0,C 180,E1 -12876.118,E2 -12876.118} C_VEL
LIN {X 0,Y 375.302,Z 250.031,A -85,B 0,C 180,E1 -12876.171,E2 -12876.171} C_VEL
LIN {X 0,Y 374.097,Z 246.37,A -85,B 0,C 180,E1 -12876.3,E2 -12876.3} C_VEL
LIN {X 0,Y 370.478,Z 241.055,A -85,B 0,C 180,E1 -12876.577,E2 -12876.577} C_VEL
LIN {X 0,Y 365.875,Z 234.724,A -85,B 0,C 180,E1 -12876.927,E2 -12876.927} C_VEL
LIN {X 0,Y 364.831,Z 232.325,A -85,B 0,C 180,E1 -12877.027,E2 -12877.027} C_VEL
LIN {X 0,Y 362.141,Z 224.377,A -85,B 0,C 180,E1 -12877.353,E2 -12877.353} C_VEL
LIN {X 0,Y 361.976,Z 224.394,A -85,B 0,C 180,E1 -12881.197,E2 -12881.197} C_VEL
LIN {X 0,Y 361.968,Z 224.398,A -85,B 0,C 180,E1 -12884.621,E2 -12884.621} C_VEL
LIN {X 0,Y 361.964,Z 224.398,A -85,B 0,C 180,E1 -12888.1,E2 -12888.1} C_VEL
LIN {X 0,Y 361.867,Z 224.408,A -85,B 0,C 180,E1 -12891.656,E2 -12891.656} C_VEL
LIN {X 0,Y 361.872,Z 224.406,A -85,B 0,C 180,E1 -12895.295,E2 -12895.295} C_VEL
LIN {X 0,Y 361.862,Z 224.407,A -85,B 0,C 180,E1 -12899.074,E2 -12899.074} C_VEL
LIN {X 0,Y 361.854,Z 224.408,A -85,B 0,C 180,E1 -12902.945,E2 -12902.945} C_VEL
LIN {X 0,Y 361.87,Z 224.411,A -85,B 0,C 180,E1 -12905.638,E2 -12905.638} C_VEL
LIN {X 0,Y 361.83,Z 224.412,A -85,B 0,C 180,E1 -12909.018,E2 -12909.018} C_VEL
LIN {X 0,Y 361.835,Z 224.411,A -85,B 0,C 180,E1 -12912.83,E2 -12912.83} C_VEL
LIN {X 0,Y 361.819,Z 224.414,A -85,B 0,C 180,E1 -12915.948,E2 -12915.948} C_VEL
LIN {X 0,Y 361.816,Z 224.418,A -85,B 0,C 180,E1 -12919.25,E2 -12919.25} C_VEL
LIN {X 0,Y 361.864,Z 224.411,A -85,B 0,C 180,E1 -12922.981,E2 -12922.981} C_VEL
LIN {X 0,Y 361.863,Z 224.409,A -85,B 0,C 180,E1 -12926.632,E2 -12926.632} C_VEL
LIN {X 0,Y 361.853,Z 224.409,A -85,B 0,C 180,E1 -12929.67,E2 -12929.67} C_VEL
LIN {X 0,Y 361.859,Z 224.408,A -85,B 0,C 180,E1 -12933.467,E2 -12933.467} C_VEL
LIN {X 0,Y 361.962,Z 224.523,A -85,B 0,C 180,E1 -12936.658,E2 -12936.658} C_VEL
LIN {X 0,Y 363.03,Z 230.372,A -85,B 0,C 180,E1 -12938.32,E2 -12938.32} C_VEL
LIN {X 0,Y 365.797,Z 241.884,A -85,B 0,C 180,E1 -12938.769,E2 -12938.769} C_VEL
LIN {X 0,Y 367.907,Z 254.505,A -85,B 0,C 180,E1 -12939.191,E2 -12939.191} C_VEL
LIN {X 0,Y 365.696,Z 339.096,A -85,B 0,C 180,E1 -12941.403,E2 -12941.403} C_VEL
LIN {X 0,Y 365.24,Z 353.007,A -85,B 0,C 180,E1 -12941.996,E2 -12941.996} C_VEL
LIN {X 0,Y 364.732,Z 365.673,A -85,B 0,C 180,E1 -12942.767,E2 -12942.767} C_VEL
LIN {X 0,Y 364.029,Z 377.951,A -85,B 0,C 180,E1 -12943.743,E2 -12943.743} C_VEL
LIN {X 0,Y 363.357,Z 389.081,A -85,B 0,C 180,E1 -12944.863,E2 -12944.863} C_VEL
LIN {X 0,Y 362.842,Z 398.564,A -85,B 0,C 180,E1 -12946.04,E2 -12946.04} C_VEL
LIN {X 0,Y 362.23,Z 407.591,A -85,B 0,C 180,E1 -12947.392,E2 -12947.392} C_VEL
LIN {X 0,Y 361.564,Z 416.764,A -85,B 0,C 180,E1 -12949.075,E2 -12949.075} C_VEL
LIN {X 0,Y 361.141,Z 424.061,A -85,B 0,C 180,E1 -12950.761,E2 -12950.761} C_VEL
LIN {X 0,Y 360.808,Z 430.764,A -85,B 0,C 180,E1 -12952.726,E2 -12952.726} C_VEL
LIN {X 0,Y 360.615,Z 435.118,A -85,B 0,C 180,E1 -12954.408,E2 -12954.408} C_VEL
LIN {X 0,Y 360.566,Z 437.358,A -85,B 0,C 180,E1 -12955.528,E2 -12955.528} C_VEL
LIN {X 0,Y 360.474,Z 439.153,A -85,B 0,C 180,E1 -12956.647,E2 -12956.647} C_VEL
LIN {X 0,Y 360.465,Z 440.509,A -85,B 0,C 180,E1 -12957.765,E2 -12957.765} C_VEL
LIN {X 0,Y 360.479,Z 441.383,A -85,B 0,C 180,E1 -12958.883,E2 -12958.883} C_VEL
LIN {X 0,Y 360.509,Z 441.838,A -85,B 0,C 180,E1 -12960,E2 -12960} C_VEL
LIN {X 0,Y 360.571,Z 441.881,A -85,B 0,C 180,E1 -12961.117,E2 -12961.117} C_VEL
LIN {X 0,Y 360.703,Z 441.47,A -85,B 0,C 180,E1 -12962.233,E2 -12962.233} C_VEL
LIN {X 0,Y 360.928,Z 440.607,A -85,B 0,C 180,E1 -12963.349,E2 -12963.349} C_VEL
LIN {X 0,Y 361.186,Z 439.334,A -85,B 0,C 180,E1 -12964.464,E2 -12964.464} C_VEL
LIN {X 0,Y 361.452,Z 436.589,A -85,B 0,C 180,E1 -12966.139,E2 -12966.139} C_VEL
LIN {X 0,Y 362.048,Z 432.755,A -85,B 0,C 180,E1 -12967.809,E2 -12967.809} C_VEL
LIN {X 0,Y 362.829,Z 427.77,A -85,B 0,C 180,E1 -12969.476,E2 -12969.476} C_VEL
LIN {X 0,Y 363.764,Z 421.462,A -85,B 0,C 180,E1 -12971.14,E2 -12971.14} C_VEL
LIN {X 0,Y 364.925,Z 413.57,A -85,B 0,C 180,E1 -12972.796,E2 -12972.796} C_VEL
LIN {X 0,Y 366.27,Z 403.792,A -85,B 0,C 180,E1 -12974.444,E2 -12974.444} C_VEL
LIN {X 0,Y 367.644,Z 393.617,A -85,B 0,C 180,E1 -12975.807,E2 -12975.807} C_VEL
LIN {X 0,Y 369.055,Z 382.336,A -85,B 0,C 180,E1 -12977.025,E2 -12977.025} C_VEL
LIN {X 0,Y 370.26,Z 370.208,A -85,B 0,C 180,E1 -12978.061,E2 -12978.061} C_VEL
LIN {X 0,Y 371.376,Z 357.519,A -85,B 0,C 180,E1 -12978.895,E2 -12978.895} C_VEL
LIN {X 0,Y 372.205,Z 344.674,A -85,B 0,C 180,E1 -12979.51,E2 -12979.51} C_VEL
LIN {X 0,Y 373.149,Z 326.089,A -85,B 0,C 180,E1 -12980.104,E2 -12980.104} C_VEL
LIN {X 0,Y 377.061,Z 260.275,A -85,B 0,C 180,E1 -12982.09,E2 -12982.09} C_VEL
LIN {X 0,Y 373.372,Z 251.868,A -85,B 0,C 180,E1 -12982.861,E2 -12982.861} C_VEL
LIN {X 0,Y 367.357,Z 240.86,A -85,B 0,C 180,E1 -12984.119,E2 -12984.119} C_VEL
LIN {X 0,Y 365.349,Z 237.1,A -85,B 0,C 180,E1 -12984.613,E2 -12984.613} C_VEL
LIN {X 0,Y 363.846,Z 231.035,A -85,B 0,C 180,E1 -12987.618,E2 -12987.618} C_VEL
LIN {X 0,Y 362.553,Z 226.603,A -85,B 0,C 180,E1 -12990.265,E2 -12990.265} C_VEL
LIN {X 0,Y 361.861,Z 224.411,A -85,B 0,C 180,E1 -12991.872,E2 -12991.872} C_VEL
LIN {X 0,Y 361.873,Z 224.411,A -85,B 0,C 180,E1 -12995.636,E2 -12995.636} C_VEL
LIN {X 0,Y 361.874,Z 224.407,A -85,B 0,C 180,E1 -12999.026,E2 -12999.026} C_VEL
LIN {X 0,Y 361.841,Z 224.413,A -85,B 0,C 180,E1 -13002.828,E2 -13002.828} C_VEL
LIN {X 0,Y 361.823,Z 224.416,A -85,B 0,C 180,E1 -13005.946,E2 -13005.946} C_VEL
LIN {X 0,Y 361.838,Z 224.414,A -85,B 0,C 180,E1 -13009.244,E2 -13009.244} C_VEL
LIN {X 0,Y 361.883,Z 224.477,A -85,B 0,C 180,E1 -13011.426,E2 -13011.426} C_VEL
LIN {X 0,Y 363.05,Z 228.407,A -85,B 0,C 180,E1 -13013.812,E2 -13013.812} C_VEL
LIN {X 0,Y 364.862,Z 234.326,A -85,B 0,C 180,E1 -13016.722,E2 -13016.722} C_VEL
LIN {X 0,Y 366.673,Z 241.428,A -85,B 0,C 180,E1 -13019.6,E2 -13019.6} C_VEL
LIN {X 0,Y 368.213,Z 248.939,A -85,B 0,C 180,E1 -13022.175,E2 -13022.175} C_VEL
LIN {X 0,Y 368.73,Z 253.643,A -85,B 0,C 180,E1 -13023.614,E2 -13023.614} C_VEL
LIN {X 0,Y 367.945,Z 258.433,A -85,B 0,C 180,E1 -13024.811,E2 -13024.811} C_VEL
LIN {X 0,Y 371.456,Z 273.276,A -85,B 0,C 180,E1 -13025.864,E2 -13025.864} C_VEL
LIN {X 0,Y 374.064,Z 287.161,A -85,B 0,C 180,E1 -13026.705,E2 -13026.705} C_VEL
LIN {X 0,Y 375.355,Z 299.608,A -85,B 0,C 180,E1 -13027.306,E2 -13027.306} C_VEL
LIN {X 0,Y 371.465,Z 371.726,A -85,B 0,C 180,E1 -13029.474,E2 -13029.474} C_VEL
LIN {X 0,Y 370.275,Z 385.377,A -85,B 0,C 180,E1 -13030.094,E2 -13030.094} C_VEL
LIN {X 0,Y 368.883,Z 398.955,A -85,B 0,C 180,E1 -13030.956,E2 -13030.956} C_VEL
LIN {X 0,Y 367.522,Z 410.394,A -85,B 0,C 180,E1 -13031.895,E2 -13031.895} C_VEL
LIN {X 0,Y 366.053,Z 422.127,A -85,B 0,C 180,E1 -13033.117,E2 -13033.117} C_VEL
LIN {X 0,Y 364.768,Z 431.804,A -85,B 0,C 180,E1 -13034.35,E2 -13034.35} C_VEL
LIN {X 0,Y 363.543,Z 440.74,A -85,B 0,C 180,E1 -13035.729,E2 -13035.729} C_VEL
LIN {X 0,Y 362.445,Z 449.514,A -85,B 0,C 180,E1 -13037.399,E2 -13037.399} C_VEL
LIN {X 0,Y 361.594,Z 456.635,A -85,B 0,C 180,E1 -13039.075,E2 -13039.075} C_VEL
LIN {X 0,Y 360.907,Z 463.225,A -85,B 0,C 180,E1 -13041.036,E2 -13041.036} C_VEL
LIN {X 0,Y 360.528,Z 467.536,A -85,B 0,C 180,E1 -13042.719,E2 -13042.719} C_VEL
LIN {X 0,Y 360.363,Z 470.759,A -85,B 0,C 180,E1 -13044.403,E2 -13044.403} C_VEL
LIN {X 0,Y 360.364,Z 472.308,A -85,B 0,C 180,E1 -13045.525,E2 -13045.525} C_VEL
LIN {X 0,Y 360.323,Z 473.432,A -85,B 0,C 180,E1 -13046.644,E2 -13046.644} C_VEL
LIN {X 0,Y 360.351,Z 474.135,A -85,B 0,C 180,E1 -13047.763,E2 -13047.763} C_VEL
LIN {X 0,Y 360.471,Z 474.362,A -85,B 0,C 180,E1 -13048.882,E2 -13048.882} C_VEL
LIN {X 0,Y 360.486,Z 474.144,A -85,B 0,C 180,E1 -13049.999,E2 -13049.999} C_VEL
LIN {X 0,Y 360.475,Z 472.609,A -85,B 0,C 180,E1 -13052.233,E2 -13052.233} C_VEL
LIN {X 0,Y 360.373,Z 471.837,A -85,B 0,C 180,E1 -13053.353,E2 -13053.353} C_VEL
LIN {X 0,Y 360.387,Z 470.63,A -85,B 0,C 180,E1 -13054.473,E2 -13054.473} C_VEL
LIN {X 0,Y 360.442,Z 468.239,A -85,B 0,C 180,E1 -13056.058,E2 -13056.058} C_VEL
LIN {X 0,Y 360.636,Z 464.467,A -85,B 0,C 180,E1 -13057.839,E2 -13057.839} C_VEL
LIN {X 0,Y 360.97,Z 459.766,A -85,B 0,C 180,E1 -13059.525,E2 -13059.525} C_VEL
LIN {X 0,Y 361.71,Z 452.696,A -85,B 0,C 180,E1 -13061.486,E2 -13061.486} C_VEL
LIN {X 0,Y 362.699,Z 445.036,A -85,B 0,C 180,E1 -13063.159,E2 -13063.159} C_VEL
LIN {X 0,Y 363.712,Z 435.788,A -85,B 0,C 180,E1 -13064.775,E2 -13064.775} C_VEL
LIN {X 0,Y 365.061,Z 425.519,A -85,B 0,C 180,E1 -13066.208,E2 -13066.208} C_VEL
LIN {X 0,Y 366.401,Z 414.304,A -85,B 0,C 180,E1 -13067.439,E2 -13067.439} C_VEL
LIN {X 0,Y 367.595,Z 403.321,A -85,B 0,C 180,E1 -13068.387,E2 -13068.387} C_VEL
LIN {X 0,Y 368.567,Z 392.255,A -85,B 0,C 180,E1 -13069.13,E2 -13069.13} C_VEL
LIN {X 0,Y 369.585,Z 379.878,A -85,B 0,C 180,E1 -13069.725,E2 -13069.725} C_VEL
LIN {X 0,Y 370.172,Z 366.934,A -85,B 0,C 180,E1 -13070.131,E2 -13070.131} C_VEL
LIN {X 0,Y 371.385,Z 297.639,A -85,B 0,C 180,E1 -13071.522,E2 -13071.522} C_VEL
LIN {X 0,Y 368.558,Z 277.369,A -85,B 0,C 180,E1 -13072.162,E2 -13072.162} C_VEL
LIN {X 0,Y 364.392,Z 253.201,A -85,B 0,C 180,E1 -13073.025,E2 -13073.025} C_VEL
LIN {X 0,Y 365.36,Z 242.914,A -85,B 0,C 180,E1 -13075.3,E2 -13075.3} C_VEL
LIN {X 0,Y 364.274,Z 236.045,A -85,B 0,C 180,E1 -13076.918,E2 -13076.918} C_VEL
LIN {X 0,Y 361.91,Z 224.407,A -85,B 0,C 180,E1 -13079.785,E2 -13079.785} C_VEL
LIN {X 0,Y 361.854,Z 224.381,A -85,B 0,C 180,E1 -13083.368,E2 -13083.368} C_VEL
LIN {X 0,Y 361.859,Z 224.41,A -85,B 0,C 180,E1 -13087.017,E2 -13087.017} C_VEL
LIN {X 0,Y 361.807,Z 224.415,A -85,B 0,C 180,E1 -13090.75,E2 -13090.75} C_VEL
LIN {X 0,Y 361.81,Z 224.412,A -85,B 0,C 180,E1 -13094.368,E2 -13094.368} C_VEL
LIN {X 0,Y 361.823,Z 224.403,A -85,B 0,C 180,E1 -13097.568,E2 -13097.568} C_VEL
LIN {X 0,Y 361.836,Z 224.412,A -85,B 0,C 180,E1 -13101.571,E2 -13101.571} C_VEL
LIN {X 0,Y 361.866,Z 224.389,A -85,B 0,C 180,E1 -13104.655,E2 -13104.655} C_VEL
LIN {X 0,Y 361.83,Z 224.407,A -85,B 0,C 180,E1 -13108.37,E2 -13108.37} C_VEL
LIN {X 0,Y 361.857,Z 224.387,A -85,B 0,C 180,E1 -13110.952,E2 -13110.952} C_VEL
LIN {X 0,Y 361.87,Z 224.405,A -85,B 0,C 180,E1 -13114.706,E2 -13114.706} C_VEL
LIN {X 0,Y 361.844,Z 224.383,A -85,B 0,C 180,E1 -13118.344,E2 -13118.344} C_VEL
LIN {X 0,Y 361.911,Z 224.4,A -85,B 0,C 180,E1 -13122.084,E2 -13122.084} C_VEL
LIN {X 0,Y 361.989,Z 224.366,A -85,B 0,C 180,E1 -13126.101,E2 -13126.101} C_VEL
LIN {X 0,Y 361.99,Z 224.392,A -85,B 0,C 180,E1 -13129.937,E2 -13129.937} C_VEL
LIN {X 0,Y 362.106,Z 224.362,A -85,B 0,C 180,E1 -13133.313,E2 -13133.313} C_VEL
LIN {X 0,Y 362.261,Z 224.354,A -85,B 0,C 180,E1 -13137.777,E2 -13137.777} C_VEL
LIN {X 0,Y 362.198,Z 224.353,A -85,B 0,C 180,E1 -13141.112,E2 -13141.112} C_VEL
LIN {X 0,Y 362.258,Z 224.334,A -85,B 0,C 180,E1 -13142.224,E2 -13142.224} C_VEL
LIN {X 0,Y 362.152,Z 224.368,A -85,B 0,C 180,E1 -13146.687,E2 -13146.687} C_VEL
LIN {X 0,Y 362.022,Z 224.366,A -85,B 0,C 180,E1 -13150.063,E2 -13150.063} C_VEL
LIN {X 0,Y 361.99,Z 224.394,A -85,B 0,C 180,E1 -13153.899,E2 -13153.899} C_VEL
LIN {X 0,Y 361.92,Z 224.385,A -85,B 0,C 180,E1 -13156.935,E2 -13156.935} C_VEL
LIN {X 0,Y 361.887,Z 224.405,A -85,B 0,C 180,E1 -13160.461,E2 -13160.461} C_VEL
LIN {X 0,Y 361.888,Z 224.393,A -85,B 0,C 180,E1 -13164.115,E2 -13164.115} C_VEL
LIN {X 0,Y 361.935,Z 224.4,A -85,B 0,C 180,E1 -13166.722,E2 -13166.722} C_VEL
LIN {X 0,Y 361.867,Z 224.404,A -85,B 0,C 180,E1 -13170.329,E2 -13170.329} C_VEL
LIN {X 0,Y 361.849,Z 224.402,A -85,B 0,C 180,E1 -13174.282,E2 -13174.282} C_VEL
LIN {X 0,Y 361.86,Z 224.41,A -85,B 0,C 180,E1 -13177.225,E2 -13177.225} C_VEL
LIN {X 0,Y 361.833,Z 224.418,A -85,B 0,C 180,E1 -13180.757,E2 -13180.757} C_VEL
LIN {X 0,Y 361.816,Z 224.415,A -85,B 0,C 180,E1 -13184.369,E2 -13184.369} C_VEL
LIN {X 0,Y 361.834,Z 224.41,A -85,B 0,C 180,E1 -13187.569,E2 -13187.569} C_VEL
LIN {X 0,Y 361.868,Z 224.41,A -85,B 0,C 180,E1 -13190.975,E2 -13190.975} C_VEL
LIN {X 0,Y 361.862,Z 224.482,A -85,B 0,C 180,E1 -13192.575,E2 -13192.575} C_VEL
LIN {X 0,Y 362.869,Z 227.285,A -85,B 0,C 180,E1 -13192.719,E2 -13192.719} C_VEL
LIN {X 0,Y 367.919,Z 237.607,A -85,B 0,C 180,E1 -13193.35,E2 -13193.35} C_VEL
LIN {X 0,Y 371.53,Z 246.28,A -85,B 0,C 180,E1 -13193.816,E2 -13193.816} C_VEL
LIN {X 0,Y 372.873,Z 254.744,A -85,B 0,C 180,E1 -13194.096,E2 -13194.096} C_VEL
LIN {X 0,Y 371.067,Z 338.092,A -85,B 0,C 180,E1 -13195.747,E2 -13195.747} C_VEL
LIN {X 0,Y 370.535,Z 350.962,A -85,B 0,C 180,E1 -13196.203,E2 -13196.203} C_VEL
LIN {X 0,Y 369.889,Z 362.194,A -85,B 0,C 180,E1 -13196.797,E2 -13196.797} C_VEL
LIN {X 0,Y 368.906,Z 373.836,A -85,B 0,C 180,E1 -13197.618,E2 -13197.618} C_VEL
LIN {X 0,Y 367.846,Z 384.881,A -85,B 0,C 180,E1 -13198.627,E2 -13198.627} C_VEL
LIN {X 0,Y 366.665,Z 394.558,A -85,B 0,C 180,E1 -13199.722,E2 -13199.722} C_VEL
LIN {X 0,Y 365.558,Z 403.466,A -85,B 0,C 180,E1 -13200.96,E2 -13200.96} C_VEL
LIN {X 0,Y 364.386,Z 412.54,A -85,B 0,C 180,E1 -13202.526,E2 -13202.526} C_VEL
LIN {X 0,Y 363.262,Z 420.349,A -85,B 0,C 180,E1 -13204.197,E2 -13204.197} C_VEL
LIN {X 0,Y 362.335,Z 426.924,A -85,B 0,C 180,E1 -13205.965,E2 -13205.965} C_VEL
LIN {X 0,Y 361.608,Z 432.026,A -85,B 0,C 180,E1 -13207.73,E2 -13207.73} C_VEL
LIN {X 0,Y 361.081,Z 435.889,A -85,B 0,C 180,E1 -13209.493,E2 -13209.493} C_VEL
LIN {X 0,Y 360.779,Z 437.847,A -85,B 0,C 180,E1 -13210.662,E2 -13210.662} C_VEL
LIN {X 0,Y 360.478,Z 440.247,A -85,B 0,C 180,E1 -13212.81,E2 -13212.81} C_VEL
LIN {X 0,Y 360.33,Z 440.99,A -85,B 0,C 180,E1 -13214.155,E2 -13214.155} C_VEL
LIN {X 0,Y 360.26,Z 441.198,A -85,B 0,C 180,E1 -13215.31,E2 -13215.31} C_VEL
LIN {X 0,Y 360.339,Z 440.576,A -85,B 0,C 180,E1 -13217.214,E2 -13217.214} C_VEL
LIN {X 0,Y 360.371,Z 439.249,A -85,B 0,C 180,E1 -13218.755,E2 -13218.755} C_VEL
LIN {X 0,Y 360.425,Z 437.749,A -85,B 0,C 180,E1 -13219.894,E2 -13219.894} C_VEL
LIN {X 0,Y 360.701,Z 434.685,A -85,B 0,C 180,E1 -13221.598,E2 -13221.598} C_VEL
LIN {X 0,Y 361.031,Z 430.561,A -85,B 0,C 180,E1 -13223.294,E2 -13223.294} C_VEL
LIN {X 0,Y 361.453,Z 424.289,A -85,B 0,C 180,E1 -13225.261,E2 -13225.261} C_VEL
LIN {X 0,Y 362.061,Z 417.42,A -85,B 0,C 180,E1 -13226.941,E2 -13226.941} C_VEL
LIN {X 0,Y 362.877,Z 408.812,A -85,B 0,C 180,E1 -13228.614,E2 -13228.614} C_VEL
LIN {X 0,Y 363.659,Z 400.02,A -85,B 0,C 180,E1 -13230.001,E2 -13230.001} C_VEL
LIN {X 0,Y 364.552,Z 390.346,A -85,B 0,C 180,E1 -13231.244,E2 -13231.244} C_VEL
LIN {X 0,Y 365.421,Z 379.666,A -85,B 0,C 180,E1 -13232.344,E2 -13232.344} C_VEL
LIN {X 0,Y 366.225,Z 367.845,A -85,B 0,C 180,E1 -13233.302,E2 -13233.302} C_VEL
LIN {X 0,Y 366.831,Z 356.39,A -85,B 0,C 180,E1 -13234.009,E2 -13234.009} C_VEL
LIN {X 0,Y 367.314,Z 343.708,A -85,B 0,C 180,E1 -13234.562,E2 -13234.562} C_VEL
LIN {X 0,Y 367.599,Z 329.543,A -85,B 0,C 180,E1 -13234.937,E2 -13234.937} C_VEL
LIN {X 0,Y 368.725,Z 252.235,A -85,B 0,C 180,E1 -13236.435,E2 -13236.435} C_VEL
LIN {X 0,Y 365.795,Z 235.474,A -85,B 0,C 180,E1 -13236.915,E2 -13236.915} C_VEL
LIN {X 0,Y 364.831,Z 232.325,A -85,B 0,C 180,E1 -13237.027,E2 -13237.027} C_VEL
LIN {X 0,Y 363.643,Z 229.685,A -85,B 0,C 180,E1 -13237.234,E2 -13237.234} C_VEL
LIN {X 0,Y 361.833,Z 227.283,A -85,B 0,C 180,E1 -13237.689,E2 -13237.689} C_VEL
LIN {X 0,Y 359.396,Z 225.504,A -85,B 0,C 180,E1 -13238.482,E2 -13238.482} C_VEL
LIN {X 0,Y 357.222,Z 225.046,A -85,B 0,C 180,E1 -13239.431,E2 -13239.431} C_VEL
LIN {X 0,Y 355.252,Z 225.234,A -85,B 0,C 180,E1 -13240.809,E2 -13240.809} C_VEL
LIN {X 0,Y 354.933,Z 225.27,A -85,B 0,C 180,E1 -13241.515,E2 -13241.515} C_VEL
LIN {X 0,Y 354.926,Z 225.273,A -85,B 0,C 180,E1 -13244.918,E2 -13244.918} C_VEL
LIN {X 0,Y 354.91,Z 225.278,A -85,B 0,C 180,E1 -13248.473,E2 -13248.473} C_VEL
LIN {X 0,Y 354.821,Z 225.289,A -85,B 0,C 180,E1 -13252.108,E2 -13252.108} C_VEL
LIN {X 0,Y 354.809,Z 225.289,A -85,B 0,C 180,E1 -13255.836,E2 -13255.836} C_VEL
LIN {X 0,Y 354.802,Z 225.29,A -85,B 0,C 180,E1 -13259.685,E2 -13259.685} C_VEL
LIN {X 0,Y 354.793,Z 225.289,A -85,B 0,C 180,E1 -13262.334,E2 -13262.334} C_VEL
LIN {X 0,Y 354.824,Z 225.289,A -85,B 0,C 180,E1 -13265.699,E2 -13265.699} C_VEL
LIN {X 0,Y 354.774,Z 225.294,A -85,B 0,C 180,E1 -13269.413,E2 -13269.413} C_VEL
LIN {X 0,Y 354.787,Z 225.289,A -85,B 0,C 180,E1 -13272.866,E2 -13272.866} C_VEL
LIN {X 0,Y 354.768,Z 225.291,A -85,B 0,C 180,E1 -13276.103,E2 -13276.103} C_VEL
LIN {X 0,Y 354.769,Z 225.295,A -85,B 0,C 180,E1 -13279.176,E2 -13279.176} C_VEL
LIN {X 0,Y 354.803,Z 225.287,A -85,B 0,C 180,E1 -13282.405,E2 -13282.405} C_VEL
LIN {X 0,Y 354.812,Z 225.29,A -85,B 0,C 180,E1 -13284.94,E2 -13284.94} C_VEL
LIN {X 0,Y 354.782,Z 225.29,A -85,B 0,C 180,E1 -13288.41,E2 -13288.41} C_VEL
LIN {X 0,Y 354.794,Z 225.288,A -85,B 0,C 180,E1 -13291.614,E2 -13291.614} C_VEL
LIN {X 0,Y 354.81,Z 225.286,A -85,B 0,C 180,E1 -13295.42,E2 -13295.42} C_VEL
LIN {X 0,Y 354.917,Z 225.42,A -85,B 0,C 180,E1 -13296.526,E2 -13296.526} C_VEL
LIN {X 0,Y 355.879,Z 230.809,A -85,B 0,C 180,E1 -13298.078,E2 -13298.078} C_VEL
LIN {X 0,Y 358.882,Z 242.777,A -85,B 0,C 180,E1 -13298.529,E2 -13298.529} C_VEL
LIN {X 0,Y 360.965,Z 255.498,A -85,B 0,C 180,E1 -13298.961,E2 -13298.961} C_VEL
LIN {X 0,Y 358.712,Z 339.062,A -85,B 0,C 180,E1 -13301.213,E2 -13301.213} C_VEL
LIN {X 0,Y 358.276,Z 352.296,A -85,B 0,C 180,E1 -13301.782,E2 -13301.782} C_VEL
LIN {X 0,Y 357.752,Z 365.249,A -85,B 0,C 180,E1 -13302.567,E2 -13302.567} C_VEL
LIN {X 0,Y 357.03,Z 377.646,A -85,B 0,C 180,E1 -13303.562,E2 -13303.562} C_VEL
LIN {X 0,Y 356.348,Z 388.923,A -85,B 0,C 180,E1 -13304.705,E2 -13304.705} C_VEL
LIN {X 0,Y 355.742,Z 399.6,A -85,B 0,C 180,E1 -13306.059,E2 -13306.059} C_VEL
LIN {X 0,Y 355.11,Z 408.455,A -85,B 0,C 180,E1 -13307.426,E2 -13307.426} C_VEL
LIN {X 0,Y 354.52,Z 416.141,A -85,B 0,C 180,E1 -13308.855,E2 -13308.855} C_VEL
LIN {X 0,Y 354.085,Z 423.676,A -85,B 0,C 180,E1 -13310.575,E2 -13310.575} C_VEL
LIN {X 0,Y 353.733,Z 430.526,A -85,B 0,C 180,E1 -13312.58,E2 -13312.58} C_VEL
LIN {X 0,Y 353.529,Z 435.025,A -85,B 0,C 180,E1 -13314.295,E2 -13314.295} C_VEL
LIN {X 0,Y 353.5,Z 437.385,A -85,B 0,C 180,E1 -13315.438,E2 -13315.438} C_VEL
LIN {X 0,Y 353.391,Z 439.24,A -85,B 0,C 180,E1 -13316.579,E2 -13316.579} C_VEL
LIN {X 0,Y 353.366,Z 440.668,A -85,B 0,C 180,E1 -13317.72,E2 -13317.72} C_VEL
LIN {X 0,Y 353.384,Z 441.652,A -85,B 0,C 180,E1 -13318.86,E2 -13318.86} C_VEL
LIN {X 0,Y 353.444,Z 442.166,A -85,B 0,C 180,E1 -13320,E2 -13320} C_VEL
LIN {X 0,Y 353.508,Z 442.268,A -85,B 0,C 180,E1 -13321.139,E2 -13321.139} C_VEL
LIN {X 0,Y 353.648,Z 441.955,A -85,B 0,C 180,E1 -13322.278,E2 -13322.278} C_VEL
LIN {X 0,Y 353.882,Z 441.17,A -85,B 0,C 180,E1 -13323.415,E2 -13323.415} C_VEL
LIN {X 0,Y 354.155,Z 439.954,A -85,B 0,C 180,E1 -13324.553,E2 -13324.553} C_VEL
LIN {X 0,Y 354.436,Z 437.336,A -85,B 0,C 180,E1 -13326.261,E2 -13326.261} C_VEL
LIN {X 0,Y 354.725,Z 435.018,A -85,B 0,C 180,E1 -13327.399,E2 -13327.399} C_VEL
LIN {X 0,Y 355.621,Z 430.55,A -85,B 0,C 180,E1 -13329.096,E2 -13329.096} C_VEL
LIN {X 0,Y 356.735,Z 423.759,A -85,B 0,C 180,E1 -13331.074,E2 -13331.074} C_VEL
LIN {X 0,Y 357.943,Z 416.372,A -85,B 0,C 180,E1 -13332.761,E2 -13332.761} C_VEL
LIN {X 0,Y 359.095,Z 408.875,A -85,B 0,C 180,E1 -13334.161,E2 -13334.161} C_VEL
LIN {X 0,Y 360.564,Z 398.778,A -85,B 0,C 180,E1 -13335.691,E2 -13335.691} C_VEL
LIN {X 0,Y 362.029,Z 388.622,A -85,B 0,C 180,E1 -13336.929,E2 -13336.929} C_VEL
LIN {X 0,Y 363.346,Z 377.564,A -85,B 0,C 180,E1 -13338.028,E2 -13338.028} C_VEL
LIN {X 0,Y 364.563,Z 365.859,A -85,B 0,C 180,E1 -13338.945,E2 -13338.945} C_VEL
LIN {X 0,Y 365.634,Z 352.854,A -85,B 0,C 180,E1 -13339.729,E2 -13339.729} C_VEL
LIN {X 0,Y 366.511,Z 339.16,A -85,B 0,C 180,E1 -13340.301,E2 -13340.301} C_VEL
LIN {X 0,Y 371.289,Z 262.44,A -85,B 0,C 180,E1 -13342.693,E2 -13342.693} C_VEL
LIN {X 0,Y 366.906,Z 253.004,A -85,B 0,C 180,E1 -13343.653,E2 -13343.653} C_VEL
LIN {X 0,Y 360.663,Z 241.81,A -85,B 0,C 180,E1 -13345.066,E2 -13345.066} C_VEL
LIN {X 0,Y 358.378,Z 237.928,A -85,B 0,C 180,E1 -13345.635,E2 -13345.635} C_VEL
LIN {X 0,Y 357.182,Z 233.185,A -85,B 0,C 180,E1 -13348.179,E2 -13348.179} C_VEL
LIN {X 0,Y 355.589,Z 227.727,A -85,B 0,C 180,E1 -13351.801,E2 -13351.801} C_VEL
LIN {X 0,Y 354.829,Z 225.287,A -85,B 0,C 180,E1 -13354.023,E2 -13354.023} C_VEL
LIN {X 0,Y 354.812,Z 225.287,A -85,B 0,C 180,E1 -13357.597,E2 -13357.597} C_VEL
LIN {X 0,Y 354.793,Z 225.29,A -85,B 0,C 180,E1 -13361.171,E2 -13361.171} C_VEL
LIN {X 0,Y 354.768,Z 225.296,A -85,B 0,C 180,E1 -13364.506,E2 -13364.506} C_VEL
LIN {X 0,Y 354.798,Z 225.292,A -85,B 0,C 180,E1 -13367.662,E2 -13367.662} C_VEL
LIN {X 0,Y 354.813,Z 225.44,A -85,B 0,C 180,E1 -13369.369,E2 -13369.369} C_VEL
LIN {X 0,Y 356.493,Z 230.456,A -85,B 0,C 180,E1 -13373.037,E2 -13373.037} C_VEL
LIN {X 0,Y 358.057,Z 235.903,A -85,B 0,C 180,E1 -13375.928,E2 -13375.928} C_VEL
LIN {X 0,Y 359.776,Z 242.552,A -85,B 0,C 180,E1 -13378.821,E2 -13378.821} C_VEL
LIN {X 0,Y 361.322,Z 249.654,A -85,B 0,C 180,E1 -13381.433,E2 -13381.433} C_VEL
LIN {X 0,Y 362.116,Z 255.165,A -85,B 0,C 180,E1 -13383.224,E2 -13383.224} C_VEL
LIN {X 0,Y 361.73,Z 257.854,A -85,B 0,C 180,E1 -13383.922,E2 -13383.922} C_VEL
LIN {X 0,Y 365.572,Z 273.57,A -85,B 0,C 180,E1 -13385.137,E2 -13385.137} C_VEL
LIN {X 0,Y 368.155,Z 287.691,A -85,B 0,C 180,E1 -13386.041,E2 -13386.041} C_VEL
LIN {X 0,Y 369.546,Z 300.013,A -85,B 0,C 180,E1 -13386.685,E2 -13386.685} C_VEL
LIN {X 0,Y 365.378,Z 371.156,A -85,B 0,C 180,E1 -13388.895,E2 -13388.895} C_VEL
LIN {X 0,Y 364.086,Z 384.741,A -85,B 0,C 180,E1 -13389.519,E2 -13389.519} C_VEL
LIN {X 0,Y 362.518,Z 399.186,A -85,B 0,C 180,E1 -13390.462,E2 -13390.462} C_VEL
LIN {X 0,Y 360.885,Z 411.806,A -85,B 0,C 180,E1 -13391.55,E2 -13391.55} C_VEL
LIN {X 0,Y 359.339,Z 423.215,A -85,B 0,C 180,E1 -13392.792,E2 -13392.792} C_VEL
LIN {X 0,Y 357.998,Z 432.609,A -85,B 0,C 180,E1 -13394.046,E2 -13394.046} C_VEL
LIN {X 0,Y 356.689,Z 441.29,A -85,B 0,C 180,E1 -13395.449,E2 -13395.449} C_VEL
LIN {X 0,Y 355.535,Z 449.88,A -85,B 0,C 180,E1 -13397.15,E2 -13397.15} C_VEL
LIN {X 0,Y 354.61,Z 456.867,A -85,B 0,C 180,E1 -13398.857,E2 -13398.857} C_VEL
LIN {X 0,Y 354.021,Z 461.611,A -85,B 0,C 180,E1 -13400.284,E2 -13400.284} C_VEL
LIN {X 0,Y 353.605,Z 466.201,A -85,B 0,C 180,E1 -13402.001,E2 -13402.001} C_VEL
LIN {X 0,Y 353.315,Z 470.226,A -85,B 0,C 180,E1 -13404.033,E2 -13404.033} C_VEL
LIN {X 0,Y 353.275,Z 472.11,A -85,B 0,C 180,E1 -13405.435,E2 -13405.435} C_VEL
LIN {X 0,Y 353.242,Z 473.19,A -85,B 0,C 180,E1 -13406.577,E2 -13406.577} C_VEL
LIN {X 0,Y 353.253,Z 473.811,A -85,B 0,C 180,E1 -13407.718,E2 -13407.718} C_VEL
LIN {X 0,Y 353.387,Z 473.98,A -85,B 0,C 180,E1 -13408.859,E2 -13408.859} C_VEL
LIN {X 0,Y 353.423,Z 473.718,A -85,B 0,C 180,E1 -13409.999,E2 -13409.999} C_VEL
LIN {X 0,Y 353.372,Z 472.32,A -85,B 0,C 180,E1 -13412.278,E2 -13412.278} C_VEL
LIN {X 0,Y 353.289,Z 471.573,A -85,B 0,C 180,E1 -13413.42,E2 -13413.42} C_VEL
LIN {X 0,Y 353.298,Z 470.402,A -85,B 0,C 180,E1 -13414.563,E2 -13414.563} C_VEL
LIN {X 0,Y 353.335,Z 468.339,A -85,B 0,C 180,E1 -13415.999,E2 -13415.999} C_VEL
LIN {X 0,Y 353.562,Z 464.322,A -85,B 0,C 180,E1 -13417.997,E2 -13417.997} C_VEL
LIN {X 0,Y 353.945,Z 459.672,A -85,B 0,C 180,E1 -13419.715,E2 -13419.715} C_VEL
LIN {X 0,Y 354.733,Z 452.66,A -85,B 0,C 180,E1 -13421.715,E2 -13421.715} C_VEL
LIN {X 0,Y 355.779,Z 445.088,A -85,B 0,C 180,E1 -13423.42,E2 -13423.42} C_VEL
LIN {X 0,Y 356.774,Z 436.507,A -85,B 0,C 180,E1 -13424.975,E2 -13424.975} C_VEL
LIN {X 0,Y 358.096,Z 426.828,A -85,B 0,C 180,E1 -13426.386,E2 -13426.386} C_VEL
LIN {X 0,Y 359.506,Z 416.121,A -85,B 0,C 180,E1 -13427.637,E2 -13427.637} C_VEL
LIN {X 0,Y 360.753,Z 405.665,A -85,B 0,C 180,E1 -13428.602,E2 -13428.602} C_VEL
LIN {X 0,Y 361.814,Z 394.226,A -85,B 0,C 180,E1 -13429.428,E2 -13429.428} C_VEL
LIN {X 0,Y 362.928,Z 381.301,A -85,B 0,C 180,E1 -13430.103,E2 -13430.103} C_VEL
LIN {X 0,Y 363.653,Z 368.146,A -85,B 0,C 180,E1 -13430.547,E2 -13430.547} C_VEL
LIN {X 0,Y 364.959,Z 298.311,A -85,B 0,C 180,E1 -13431.98,E2 -13431.98} C_VEL
LIN {X 0,Y 362.275,Z 278.994,A -85,B 0,C 180,E1 -13432.608,E2 -13432.608} C_VEL
LIN {X 0,Y 357.56,Z 251.839,A -85,B 0,C 180,E1 -13433.596,E2 -13433.596} C_VEL
LIN {X 0,Y 358.296,Z 243.132,A -85,B 0,C 180,E1 -13435.563,E2 -13435.563} C_VEL
